   IF #_w5 AND ("DB_Data".F20.Sensor_Correct_Position OR ("DB_Data".F19.Sensor_Correct_Position AND NOT "DB_Data".F20.Btt_Down_Selected) OR ("DB_Data".F18.Sensor_Correct_Position AND NOT "DB_Data".F20.Btt_Down_Selected AND NOT "DB_Data".F19.Btt_Up_Selected AND NOT "DB_Data".F19.Btt_Down_Selected) OR ("DB_Data".F17.Sensor_Correct_Position AND NOT "DB_Data".F20.Btt_Down_Selected AND NOT "DB_Data".F19.Btt_Up_Selected AND NOT "DB_Data".F19.Btt_Down_Selected AND NOT "DB_Data".F18.Btt_Up_Selected AND NOT "DB_Data".F18.Btt_Down_Selected) OR ("DB_Data".F16.Sensor_Correct_Position AND NOT "DB_Data".F20.Btt_Down_Selected AND NOT "DB_Data".F19.Btt_Up_Selected AND NOT "DB_Data".F19.Btt_Down_Selected AND NOT "DB_Data".F18.Btt_Up_Selected AND NOT "DB_Data".F18.Btt_Down_Selected AND NOT "DB_Data".F17.Btt_Up_Selected AND NOT "DB_Data".F17.Btt_Down_Selected) OR ("DB_Data".F15.Sensor_Correct_Position AND NOT "DB_Data".F20.Btt_Down_Selected AND NOT "DB_Data".F19.Btt_Up_Selected AND NOT "DB_Data".F19.Btt_Down_Selected AND NOT "DB_Data".F18.Btt_Up_Selected AND NOT "DB_Data".F18.Btt_Down_Selected AND NOT "DB_Data".F17.Btt_Up_Selected AND NOT "DB_Data".F17.Btt_Down_Selected AND NOT "DB_Data".F16.Btt_Up_Selected AND NOT "DB_Data".F16.Btt_Down_Selected) OR ("DB_Data".F14.Sensor_Correct_Position AND NOT "DB_Data".F20.Btt_Down_Selected AND NOT "DB_Data".F19.Btt_Up_Selected AND NOT "DB_Data".F19.Btt_Down_Selected AND NOT "DB_Data".F18.Btt_Up_Selected AND NOT "DB_Data".F18.Btt_Down_Selected AND NOT "DB_Data".F17.Btt_Up_Selected AND NOT "DB_Data".F17.Btt_Down_Selected AND NOT "DB_Data".F16.Btt_Up_Selected AND NOT "DB_Data".F16.Btt_Down_Selected AND NOT "DB_Data".F15.Btt_Up_Selected AND NOT "DB_Data".F15.Btt_Down_Selected) OR ("DB_Data".F13.Sensor_Correct_Position AND NOT "DB_Data".F20.Btt_Down_Selected AND NOT "DB_Data".F19.Btt_Up_Selected AND NOT "DB_Data".F19.Btt_Down_Selected AND NOT "DB_Data".F18.Btt_Up_Selected AND NOT "DB_Data".F18.Btt_Down_Selected AND NOT "DB_Data".F17.Btt_Up_Selected AND NOT "DB_Data".F17.Btt_Down_Selected AND NOT "DB_Data".F16.Btt_Up_Selected AND NOT "DB_Data".F16.Btt_Down_Selected AND NOT "DB_Data".F15.Btt_Up_Selected AND NOT "DB_Data".F15.Btt_Down_Selected AND NOT "DB_Data".F14.Btt_Up_Selected AND NOT "DB_Data".F14.Btt_Down_Selected) OR ("DB_Data".F12.Sensor_Correct_Position AND NOT "DB_Data".F20.Btt_Down_Selected AND NOT "DB_Data".F19.Btt_Up_Selected AND NOT "DB_Data".F19.Btt_Down_Selected AND NOT "DB_Data".F18.Btt_Up_Selected AND NOT "DB_Data".F18.Btt_Down_Selected AND NOT "DB_Data".F17.Btt_Up_Selected AND NOT "DB_Data".F17.Btt_Down_Selected AND NOT "DB_Data".F16.Btt_Up_Selected AND NOT "DB_Data".F16.Btt_Down_Selected AND NOT "DB_Data".F15.Btt_Up_Selected AND NOT "DB_Data".F15.Btt_Down_Selected AND NOT "DB_Data".F14.Btt_Up_Selected AND NOT "DB_Data".F14.Btt_Down_Selected AND NOT "DB_Data".F13.Btt_Up_Selected AND NOT "DB_Data".F13.Btt_Down_Selected) OR ("DB_Data".F11.Sensor_Correct_Position AND NOT "DB_Data".F20.Btt_Down_Selected AND NOT "DB_Data".F19.Btt_Up_Selected AND NOT "DB_Data".F19.Btt_Down_Selected AND NOT "DB_Data".F18.Btt_Up_Selected AND NOT "DB_Data".F18.Btt_Down_Selected AND NOT "DB_Data".F17.Btt_Up_Selected AND NOT "DB_Data".F17.Btt_Down_Selected AND NOT "DB_Data".F16.Btt_Up_Selected AND NOT "DB_Data".F16.Btt_Down_Selected AND NOT "DB_Data".F15.Btt_Up_Selected AND NOT "DB_Data".F15.Btt_Down_Selected AND NOT "DB_Data".F14.Btt_Up_Selected AND NOT "DB_Data".F14.Btt_Down_Selected AND NOT "DB_Data".F13.Btt_Up_Selected AND NOT "DB_Data".F13.Btt_Down_Selected AND NOT "DB_Data".F12.Btt_Up_Selected AND NOT "DB_Data".F12.Btt_Down_Selected) OR ("DB_Data".F10.Sensor_Correct_Position AND NOT "DB_Data".F20.Btt_Down_Selected AND NOT "DB_Data".F19.Btt_Up_Selected AND NOT "DB_Data".F19.Btt_Down_Selected AND NOT "DB_Data".F18.Btt_Up_Selected AND NOT "DB_Data".F18.Btt_Down_Selected AND NOT "DB_Data".F17.Btt_Up_Selected AND NOT "DB_Data".F17.Btt_Down_Selected AND NOT "DB_Data".F16.Btt_Up_Selected AND NOT "DB_Data".F16.Btt_Down_Selected AND NOT "DB_Data".F15.Btt_Up_Selected AND NOT "DB_Data".F15.Btt_Down_Selected AND NOT "DB_Data".F14.Btt_Up_Selected AND NOT "DB_Data".F14.Btt_Down_Selected AND NOT "DB_Data".F13.Btt_Up_Selected AND NOT "DB_Data".F13.Btt_Down_Selected AND NOT "DB_Data".F12.Btt_Up_Selected AND NOT "DB_Data".F12.Btt_Down_Selected AND NOT "DB_Data".F11.Btt_Up_Selected AND NOT "DB_Data".F11.Btt_Down_Selected) OR ("DB_Data".F9.Sensor_Correct_Position AND NOT "DB_Data".F20.Btt_Down_Selected AND NOT "DB_Data".F19.Btt_Up_Selected AND NOT "DB_Data".F19.Btt_Down_Selected AND NOT "DB_Data".F18.Btt_Up_Selected AND NOT "DB_Data".F18.Btt_Down_Selected AND NOT "DB_Data".F17.Btt_Up_Selected AND NOT "DB_Data".F17.Btt_Down_Selected AND NOT "DB_Data".F16.Btt_Up_Selected AND NOT "DB_Data".F16.Btt_Down_Selected AND NOT "DB_Data".F15.Btt_Up_Selected AND NOT "DB_Data".F15.Btt_Down_Selected AND NOT "DB_Data".F14.Btt_Up_Selected AND NOT "DB_Data".F14.Btt_Down_Selected AND NOT "DB_Data".F13.Btt_Up_Selected AND NOT "DB_Data".F13.Btt_Down_Selected AND NOT "DB_Data".F12.Btt_Up_Selected AND NOT "DB_Data".F12.Btt_Down_Selected AND NOT "DB_Data".F11.Btt_Up_Selected AND NOT "DB_Data".F11.Btt_Down_Selected AND NOT "DB_Data".F10.Btt_Up_Selected AND NOT "DB_Data".F10.Btt_Down_Selected) OR ("DB_Data".F8.Sensor_Correct_Position AND NOT "DB_Data".F20.Btt_Down_Selected AND NOT "DB_Data".F19.Btt_Up_Selected AND NOT "DB_Data".F19.Btt_Down_Selected AND NOT "DB_Data".F18.Btt_Up_Selected AND NOT "DB_Data".F18.Btt_Down_Selected AND NOT "DB_Data".F17.Btt_Up_Selected AND NOT "DB_Data".F17.Btt_Down_Selected AND NOT "DB_Data".F16.Btt_Up_Selected AND NOT "DB_Data".F16.Btt_Down_Selected AND NOT "DB_Data".F15.Btt_Up_Selected AND NOT "DB_Data".F15.Btt_Down_Selected AND NOT "DB_Data".F14.Btt_Up_Selected AND NOT "DB_Data".F14.Btt_Down_Selected AND NOT "DB_Data".F13.Btt_Up_Selected AND NOT "DB_Data".F13.Btt_Down_Selected AND NOT "DB_Data".F12.Btt_Up_Selected AND NOT "DB_Data".F12.Btt_Down_Selected AND NOT "DB_Data".F11.Btt_Up_Selected AND NOT "DB_Data".F11.Btt_Down_Selected AND NOT "DB_Data".F10.Btt_Up_Selected AND NOT "DB_Data".F10.Btt_Down_Selected AND NOT "DB_Data".F9.Btt_Up_Selected AND NOT "DB_Data".F9.Btt_Down_Selected) OR ("DB_Data".F7.Sensor_Correct_Position AND NOT "DB_Data".F20.Btt_Down_Selected AND NOT "DB_Data".F19.Btt_Up_Selected AND NOT "DB_Data".F19.Btt_Down_Selected AND NOT "DB_Data".F18.Btt_Up_Selected AND NOT "DB_Data".F18.Btt_Down_Selected AND NOT "DB_Data".F17.Btt_Up_Selected AND NOT "DB_Data".F17.Btt_Down_Selected AND NOT "DB_Data".F16.Btt_Up_Selected AND NOT "DB_Data".F16.Btt_Down_Selected AND NOT "DB_Data".F15.Btt_Up_Selected AND NOT "DB_Data".F15.Btt_Down_Selected AND NOT "DB_Data".F14.Btt_Up_Selected AND NOT "DB_Data".F14.Btt_Down_Selected AND NOT "DB_Data".F13.Btt_Up_Selected AND NOT "DB_Data".F13.Btt_Down_Selected AND NOT "DB_Data".F12.Btt_Up_Selected AND NOT "DB_Data".F12.Btt_Down_Selected AND NOT "DB_Data".F11.Btt_Up_Selected AND NOT "DB_Data".F11.Btt_Down_Selected AND NOT "DB_Data".F10.Btt_Up_Selected AND NOT "DB_Data".F10.Btt_Down_Selected AND NOT "DB_Data".F9.Btt_Up_Selected AND NOT "DB_Data".F9.Btt_Down_Selected AND NOT "DB_Data".F8.Btt_Up_Selected AND NOT "DB_Data".F8.Btt_Down_Selected) OR ("DB_Data".F6.Sensor_Correct_Position AND NOT "DB_Data".F20.Btt_Down_Selected AND NOT "DB_Data".F19.Btt_Up_Selected AND NOT "DB_Data".F19.Btt_Down_Selected AND NOT "DB_Data".F18.Btt_Up_Selected AND NOT "DB_Data".F18.Btt_Down_Selected AND NOT "DB_Data".F17.Btt_Up_Selected AND NOT "DB_Data".F17.Btt_Down_Selected AND NOT "DB_Data".F16.Btt_Up_Selected AND NOT "DB_Data".F16.Btt_Down_Selected AND NOT "DB_Data".F15.Btt_Up_Selected AND NOT "DB_Data".F15.Btt_Down_Selected AND NOT "DB_Data".F14.Btt_Up_Selected AND NOT "DB_Data".F14.Btt_Down_Selected AND NOT "DB_Data".F13.Btt_Up_Selected AND NOT "DB_Data".F13.Btt_Down_Selected AND NOT "DB_Data".F12.Btt_Up_Selected AND NOT "DB_Data".F12.Btt_Down_Selected AND NOT "DB_Data".F11.Btt_Up_Selected AND NOT "DB_Data".F11.Btt_Down_Selected AND NOT "DB_Data".F10.Btt_Up_Selected AND NOT "DB_Data".F10.Btt_Down_Selected AND NOT "DB_Data".F9.Btt_Up_Selected AND NOT "DB_Data".F9.Btt_Down_Selected AND NOT "DB_Data".F8.Btt_Up_Selected AND NOT "DB_Data".F8.Btt_Down_Selected AND NOT "DB_Data".F7.Btt_Up_Selected AND NOT "DB_Data".F7.Btt_Down_Selected) OR ("DB_Data".F5.Sensor_Correct_Position AND NOT "DB_Data".F20.Btt_Down_Selected AND NOT "DB_Data".F19.Btt_Up_Selected AND NOT "DB_Data".F19.Btt_Down_Selected AND NOT "DB_Data".F18.Btt_Up_Selected AND NOT "DB_Data".F18.Btt_Down_Selected AND NOT "DB_Data".F17.Btt_Up_Selected AND NOT "DB_Data".F17.Btt_Down_Selected AND NOT "DB_Data".F16.Btt_Up_Selected AND NOT "DB_Data".F16.Btt_Down_Selected AND NOT "DB_Data".F15.Btt_Up_Selected AND NOT "DB_Data".F15.Btt_Down_Selected AND NOT "DB_Data".F14.Btt_Up_Selected AND NOT "DB_Data".F14.Btt_Down_Selected AND NOT "DB_Data".F13.Btt_Up_Selected AND NOT "DB_Data".F13.Btt_Down_Selected AND NOT "DB_Data".F12.Btt_Up_Selected AND NOT "DB_Data".F12.Btt_Down_Selected AND NOT "DB_Data".F11.Btt_Up_Selected AND NOT "DB_Data".F11.Btt_Down_Selected AND NOT "DB_Data".F10.Btt_Up_Selected AND NOT "DB_Data".F10.Btt_Down_Selected AND NOT "DB_Data".F9.Btt_Up_Selected AND NOT "DB_Data".F9.Btt_Down_Selected AND NOT "DB_Data".F8.Btt_Up_Selected AND NOT "DB_Data".F8.Btt_Down_Selected AND NOT "DB_Data".F7.Btt_Up_Selected AND NOT "DB_Data".F7.Btt_Down_Selected AND NOT "DB_Data".F6.Btt_Up_Selected AND NOT "DB_Data".F6.Btt_Down_Selected) OR ("DB_Data".F4.Sensor_Correct_Position AND NOT "DB_Data".F20.Btt_Down_Selected AND NOT "DB_Data".F19.Btt_Up_Selected AND NOT "DB_Data".F19.Btt_Down_Selected AND NOT "DB_Data".F18.Btt_Up_Selected AND NOT "DB_Data".F18.Btt_Down_Selected AND NOT "DB_Data".F17.Btt_Up_Selected AND NOT "DB_Data".F17.Btt_Down_Selected AND NOT "DB_Data".F16.Btt_Up_Selected AND NOT "DB_Data".F16.Btt_Down_Selected AND NOT "DB_Data".F15.Btt_Up_Selected AND NOT "DB_Data".F15.Btt_Down_Selected AND NOT "DB_Data".F14.Btt_Up_Selected AND NOT "DB_Data".F14.Btt_Down_Selected AND NOT "DB_Data".F13.Btt_Up_Selected AND NOT "DB_Data".F13.Btt_Down_Selected AND NOT "DB_Data".F12.Btt_Up_Selected AND NOT "DB_Data".F12.Btt_Down_Selected AND NOT "DB_Data".F11.Btt_Up_Selected AND NOT "DB_Data".F11.Btt_Down_Selected AND NOT "DB_Data".F10.Btt_Up_Selected AND NOT "DB_Data".F10.Btt_Down_Selected AND NOT "DB_Data".F9.Btt_Up_Selected AND NOT "DB_Data".F9.Btt_Down_Selected AND NOT "DB_Data".F8.Btt_Up_Selected AND NOT "DB_Data".F8.Btt_Down_Selected AND NOT "DB_Data".F7.Btt_Up_Selected AND NOT "DB_Data".F7.Btt_Down_Selected AND NOT "DB_Data".F6.Btt_Up_Selected AND NOT "DB_Data".F6.Btt_Down_Selected AND NOT "DB_Data".F5.Btt_Up_Selected AND NOT "DB_Data".F5.Btt_Down_Selected) OR ("DB_Data".F3.Sensor_Correct_Position AND NOT "DB_Data".F20.Btt_Down_Selected AND NOT "DB_Data".F19.Btt_Up_Selected AND NOT "DB_Data".F19.Btt_Down_Selected AND NOT "DB_Data".F18.Btt_Up_Selected AND NOT "DB_Data".F18.Btt_Down_Selected AND NOT "DB_Data".F17.Btt_Up_Selected AND NOT "DB_Data".F17.Btt_Down_Selected AND NOT "DB_Data".F16.Btt_Up_Selected AND NOT "DB_Data".F16.Btt_Down_Selected AND NOT "DB_Data".F15.Btt_Up_Selected AND NOT "DB_Data".F15.Btt_Down_Selected AND NOT "DB_Data".F14.Btt_Up_Selected AND NOT "DB_Data".F14.Btt_Down_Selected AND NOT "DB_Data".F13.Btt_Up_Selected AND NOT "DB_Data".F13.Btt_Down_Selected AND NOT "DB_Data".F12.Btt_Up_Selected AND NOT "DB_Data".F12.Btt_Down_Selected AND NOT "DB_Data".F11.Btt_Up_Selected AND NOT "DB_Data".F11.Btt_Down_Selected AND NOT "DB_Data".F10.Btt_Up_Selected AND NOT "DB_Data".F10.Btt_Down_Selected AND NOT "DB_Data".F9.Btt_Up_Selected AND NOT "DB_Data".F9.Btt_Down_Selected AND NOT "DB_Data".F8.Btt_Up_Selected AND NOT "DB_Data".F8.Btt_Down_Selected AND NOT "DB_Data".F7.Btt_Up_Selected AND NOT "DB_Data".F7.Btt_Down_Selected AND NOT "DB_Data".F6.Btt_Up_Selected AND NOT "DB_Data".F6.Btt_Down_Selected AND NOT "DB_Data".F5.Btt_Up_Selected AND NOT "DB_Data".F5.Btt_Down_Selected AND NOT "DB_Data".F4.Btt_Up_Selected AND NOT "DB_Data".F4.Btt_Down_Selected) OR ("DB_Data".F2.Sensor_Correct_Position AND NOT "DB_Data".F20.Btt_Down_Selected AND NOT "DB_Data".F19.Btt_Up_Selected AND NOT "DB_Data".F19.Btt_Down_Selected AND NOT "DB_Data".F18.Btt_Up_Selected AND NOT "DB_Data".F18.Btt_Down_Selected AND NOT "DB_Data".F17.Btt_Up_Selected AND NOT "DB_Data".F17.Btt_Down_Selected AND NOT "DB_Data".F16.Btt_Up_Selected AND NOT "DB_Data".F16.Btt_Down_Selected AND NOT "DB_Data".F15.Btt_Up_Selected AND NOT "DB_Data".F15.Btt_Down_Selected AND NOT "DB_Data".F14.Btt_Up_Selected AND NOT "DB_Data".F14.Btt_Down_Selected AND NOT "DB_Data".F13.Btt_Up_Selected AND NOT "DB_Data".F13.Btt_Down_Selected AND NOT "DB_Data".F12.Btt_Up_Selected AND NOT "DB_Data".F12.Btt_Down_Selected AND NOT "DB_Data".F11.Btt_Up_Selected AND NOT "DB_Data".F11.Btt_Down_Selected AND NOT "DB_Data".F10.Btt_Up_Selected AND NOT "DB_Data".F10.Btt_Down_Selected AND NOT "DB_Data".F9.Btt_Up_Selected AND NOT "DB_Data".F9.Btt_Down_Selected AND NOT "DB_Data".F8.Btt_Up_Selected AND NOT "DB_Data".F8.Btt_Down_Selected AND NOT "DB_Data".F7.Btt_Up_Selected AND NOT "DB_Data".F7.Btt_Down_Selected AND NOT "DB_Data".F6.Btt_Up_Selected AND NOT "DB_Data".F6.Btt_Down_Selected AND NOT "DB_Data".F5.Btt_Up_Selected AND NOT "DB_Data".F5.Btt_Down_Selected AND NOT "DB_Data".F4.Btt_Up_Selected AND NOT "DB_Data".F4.Btt_Down_Selected AND NOT "DB_Data".F3.Btt_Down_Selected AND NOT "DB_Data".F3.Btt_Up_Selected) OR ("DB_Data".F1.Sensor_Correct_Position AND NOT "DB_Data".F20.Btt_Down_Selected AND NOT "DB_Data".F19.Btt_Up_Selected AND NOT "DB_Data".F19.Btt_Down_Selected AND NOT "DB_Data".F18.Btt_Up_Selected AND NOT "DB_Data".F18.Btt_Down_Selected AND NOT "DB_Data".F17.Btt_Up_Selected AND NOT "DB_Data".F17.Btt_Down_Selected AND NOT "DB_Data".F16.Btt_Up_Selected AND NOT "DB_Data".F16.Btt_Down_Selected AND NOT "DB_Data".F15.Btt_Up_Selected AND NOT "DB_Data".F15.Btt_Down_Selected AND NOT "DB_Data".F14.Btt_Up_Selected AND NOT "DB_Data".F14.Btt_Down_Selected AND NOT "DB_Data".F13.Btt_Up_Selected AND NOT "DB_Data".F13.Btt_Down_Selected AND NOT "DB_Data".F12.Btt_Up_Selected AND NOT "DB_Data".F12.Btt_Down_Selected AND NOT "DB_Data".F11.Btt_Up_Selected AND NOT "DB_Data".F11.Btt_Down_Selected AND NOT "DB_Data".F10.Btt_Up_Selected AND NOT "DB_Data".F10.Btt_Down_Selected AND NOT "DB_Data".F9.Btt_Up_Selected AND NOT "DB_Data".F9.Btt_Down_Selected AND NOT "DB_Data".F8.Btt_Up_Selected AND NOT "DB_Data".F8.Btt_Down_Selected AND NOT "DB_Data".F7.Btt_Up_Selected AND NOT "DB_Data".F7.Btt_Down_Selected AND NOT "DB_Data".F6.Btt_Up_Selected AND NOT "DB_Data".F6.Btt_Down_Selected AND NOT "DB_Data".F5.Btt_Up_Selected AND NOT "DB_Data".F5.Btt_Down_Selected AND NOT "DB_Data".F4.Btt_Up_Selected AND NOT "DB_Data".F4.Btt_Down_Selected AND NOT "DB_Data".F3.Btt_Down_Selected AND NOT "DB_Data".F3.Btt_Up_Selected AND NOT "DB_Data".F2.Btt_Down_Selected AND NOT "DB_Data".F2.Btt_Up_Selected)) THEN
       "DB_Data".Last_Is_Up := FALSE;
   END_IF;
END_REGION

REGION Network 23
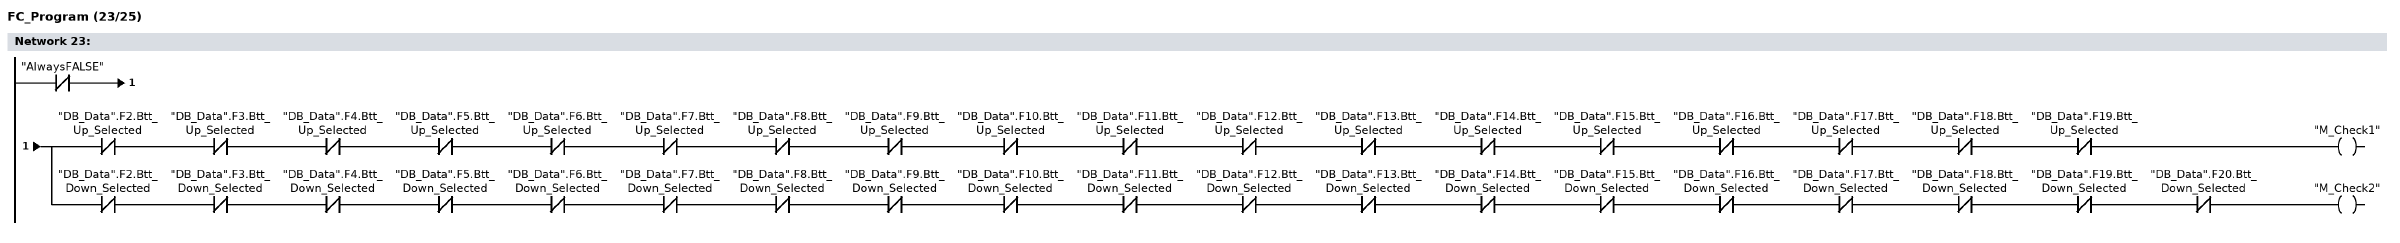
   RUNG wire#powerrail
      I_Contact( "AlwaysFALSE" )
      wire#w1
      I_Contact( "DB_Data".F2.Btt_Up_Selected )
      I_Contact( "DB_Data".F3.Btt_Up_Selected )
      I_Contact( "DB_Data".F4.Btt_Up_Selected )
      I_Contact( "DB_Data".F5.Btt_Up_Selected )
      I_Contact( "DB_Data".F6.Btt_Up_Selected )
      I_Contact( "DB_Data".F7.Btt_Up_Selected )
      I_Contact( "DB_Data".F8.Btt_Up_Selected )
      I_Contact( "DB_Data".F9.Btt_Up_Selected )
      I_Contact( "DB_Data".F10.Btt_Up_Selected )
      I_Contact( "DB_Data".F11.Btt_Up_Selected )
      I_Contact( "DB_Data".F12.Btt_Up_Selected )
      I_Contact( "DB_Data".F13.Btt_Up_Selected )
      I_Contact( "DB_Data".F14.Btt_Up_Selected )
      I_Contact( "DB_Data".F15.Btt_Up_Selected )
      I_Contact( "DB_Data".F16.Btt_Up_Selected )
      I_Contact( "DB_Data".F17.Btt_Up_Selected )
      I_Contact( "DB_Data".F18.Btt_Up_Selected )
      I_Contact( "DB_Data".F19.Btt_Up_Selected )
      Coil( "M_Check1" )
   END_RUNG
   RUNG wire#w1
      I_Contact( "DB_Data".F2.Btt_Down_Selected )
      I_Contact( "DB_Data".F3.Btt_Down_Selected )
      I_Contact( "DB_Data".F4.Btt_Down_Selected )
      I_Contact( "DB_Data".F5.Btt_Down_Selected )
      I_Contact( "DB_Data".F6.Btt_Down_Selected )
      I_Contact( "DB_Data".F7.Btt_Down_Selected )
      I_Contact( "DB_Data".F8.Btt_Down_Selected )
      I_Contact( "DB_Data".F9.Btt_Down_Selected )
      I_Contact( "DB_Data".F10.Btt_Down_Selected )
      I_Contact( "DB_Data".F11.Btt_Down_Selected )
      I_Contact( "DB_Data".F12.Btt_Down_Selected )
      I_Contact( "DB_Data".F13.Btt_Down_Selected )
      I_Contact( "DB_Data".F14.Btt_Down_Selected )
      I_Contact( "DB_Data".F15.Btt_Down_Selected )
      I_Contact( "DB_Data".F16.Btt_Down_Selected )
      I_Contact( "DB_Data".F17.Btt_Down_Selected )
      I_Contact( "DB_Data".F18.Btt_Down_Selected )
      I_Contact( "DB_Data".F19.Btt_Down_Selected )
      I_Contact( "DB_Data".F20.Btt_Down_Selected )
      Coil( "M_Check2" )
   END_RUNG
   // the same network as SCL:
   "M_Check1" := NOT "AlwaysFALSE" AND NOT "DB_Data".F2.Btt_Up_Selected AND NOT "DB_Data".F3.Btt_Up_Selected AND NOT "DB_Data".F4.Btt_Up_Selected AND NOT "DB_Data".F5.Btt_Up_Selected AND NOT "DB_Data".F6.Btt_Up_Selected AND NOT "DB_Data".F7.Btt_Up_Selected AND NOT "DB_Data".F8.Btt_Up_Selected AND NOT "DB_Data".F9.Btt_Up_Selected AND NOT "DB_Data".F10.Btt_Up_Selected AND NOT "DB_Data".F11.Btt_Up_Selected AND NOT "DB_Data".F12.Btt_Up_Selected AND NOT "DB_Data".F13.Btt_Up_Selected AND NOT "DB_Data".F14.Btt_Up_Selected AND NOT "DB_Data".F15.Btt_Up_Selected AND NOT "DB_Data".F16.Btt_Up_Selected AND NOT "DB_Data".F17.Btt_Up_Selected AND NOT "DB_Data".F18.Btt_Up_Selected AND NOT "DB_Data".F19.Btt_Up_Selected;
   "M_Check2" := NOT "AlwaysFALSE" AND NOT "DB_Data".F2.Btt_Down_Selected AND NOT "DB_Data".F3.Btt_Down_Selected AND NOT "DB_Data".F4.Btt_Down_Selected AND NOT "DB_Data".F5.Btt_Down_Selected AND NOT "DB_Data".F6.Btt_Down_Selected AND NOT "DB_Data".F7.Btt_Down_Selected AND NOT "DB_Data".F8.Btt_Down_Selected AND NOT "DB_Data".F9.Btt_Down_Selected AND NOT "DB_Data".F10.Btt_Down_Selected AND NOT "DB_Data".F11.Btt_Down_Selected AND NOT "DB_Data".F12.Btt_Down_Selected AND NOT "DB_Data".F13.Btt_Down_Selected AND NOT "DB_Data".F14.Btt_Down_Selected AND NOT "DB_Data".F15.Btt_Down_Selected AND NOT "DB_Data".F16.Btt_Down_Selected AND NOT "DB_Data".F17.Btt_Down_Selected AND NOT "DB_Data".F18.Btt_Down_Selected AND NOT "DB_Data".F19.Btt_Down_Selected AND NOT "DB_Data".F20.Btt_Down_Selected;
END_REGION

REGION Network 24: Tự động mở cửa
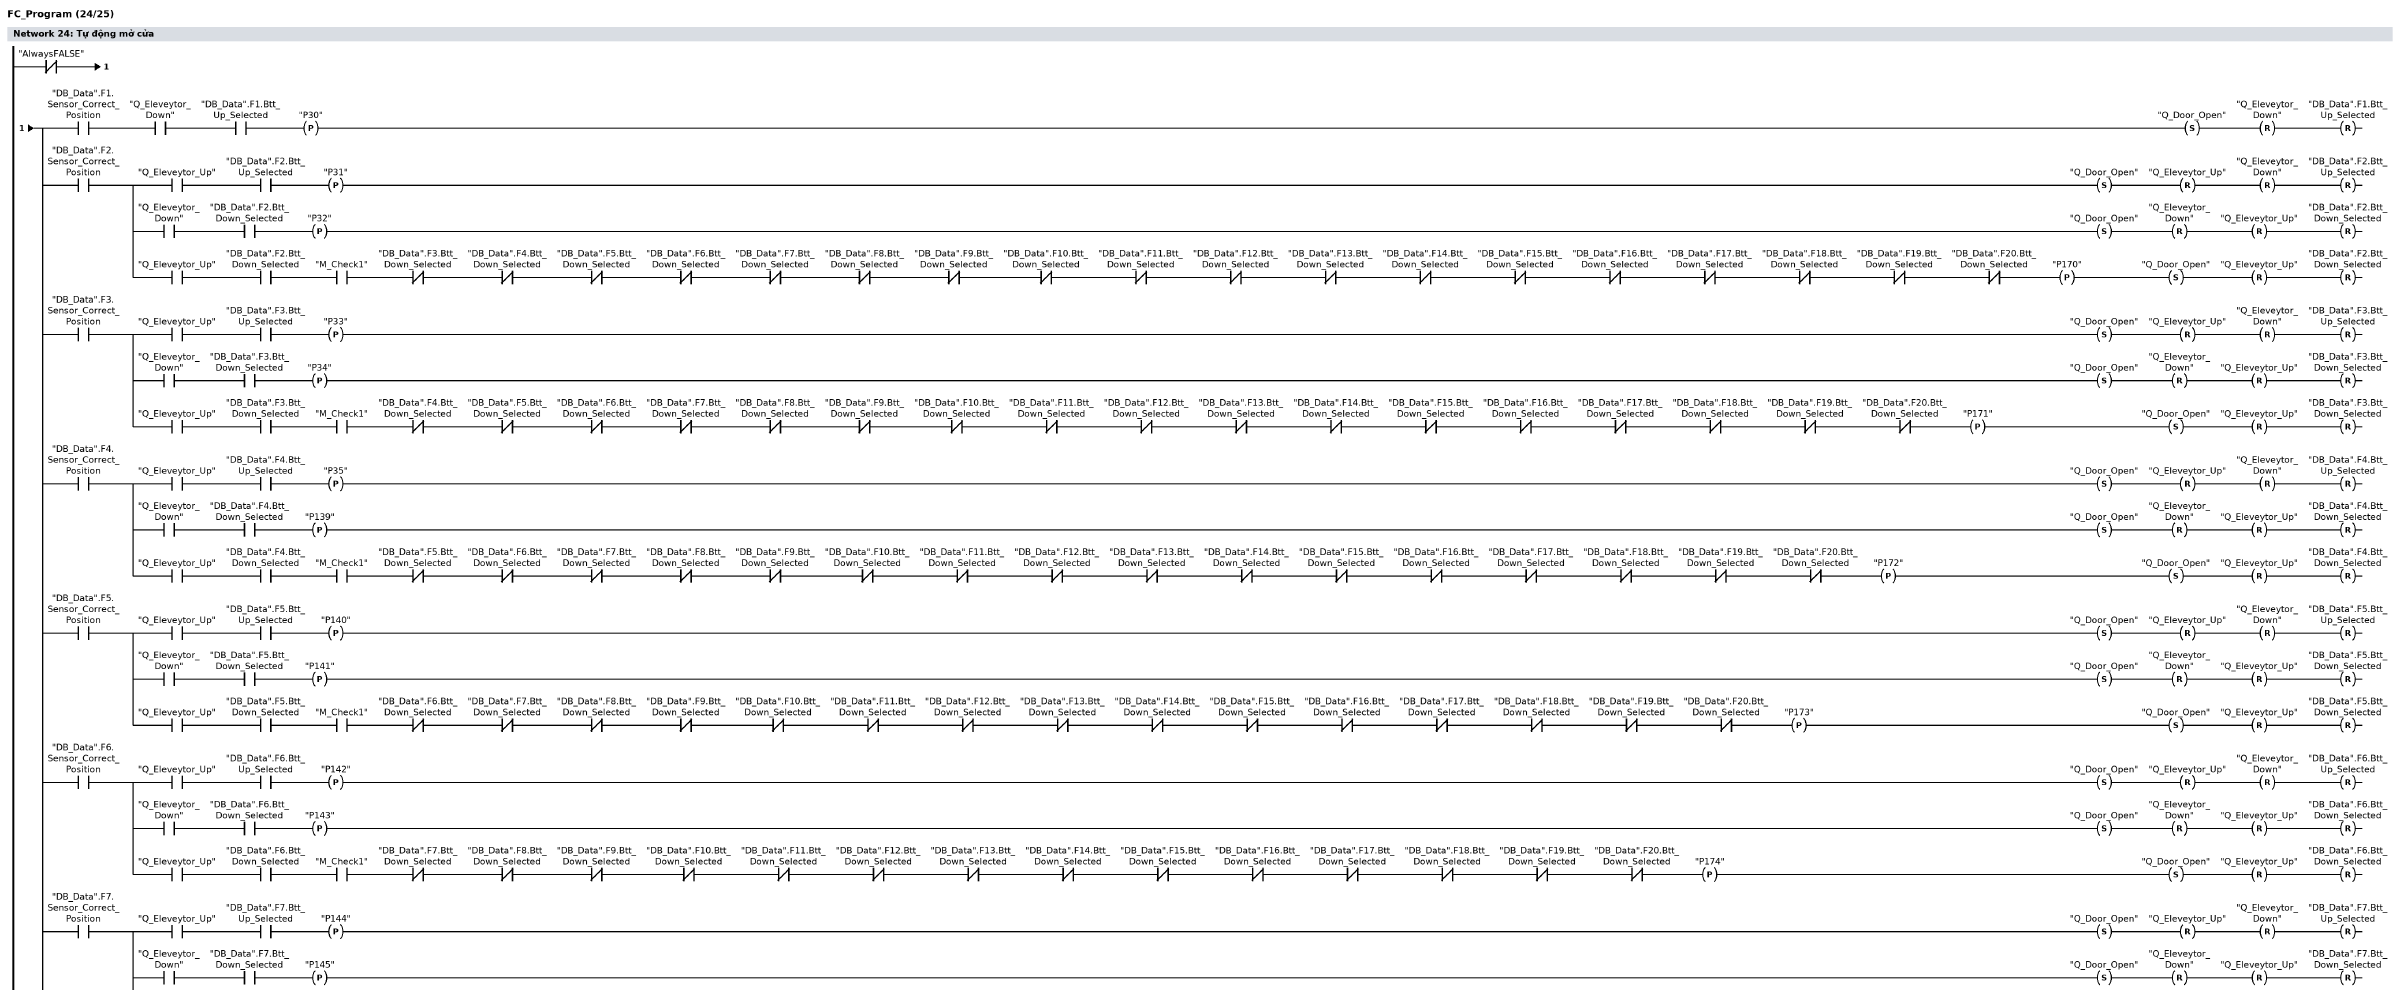
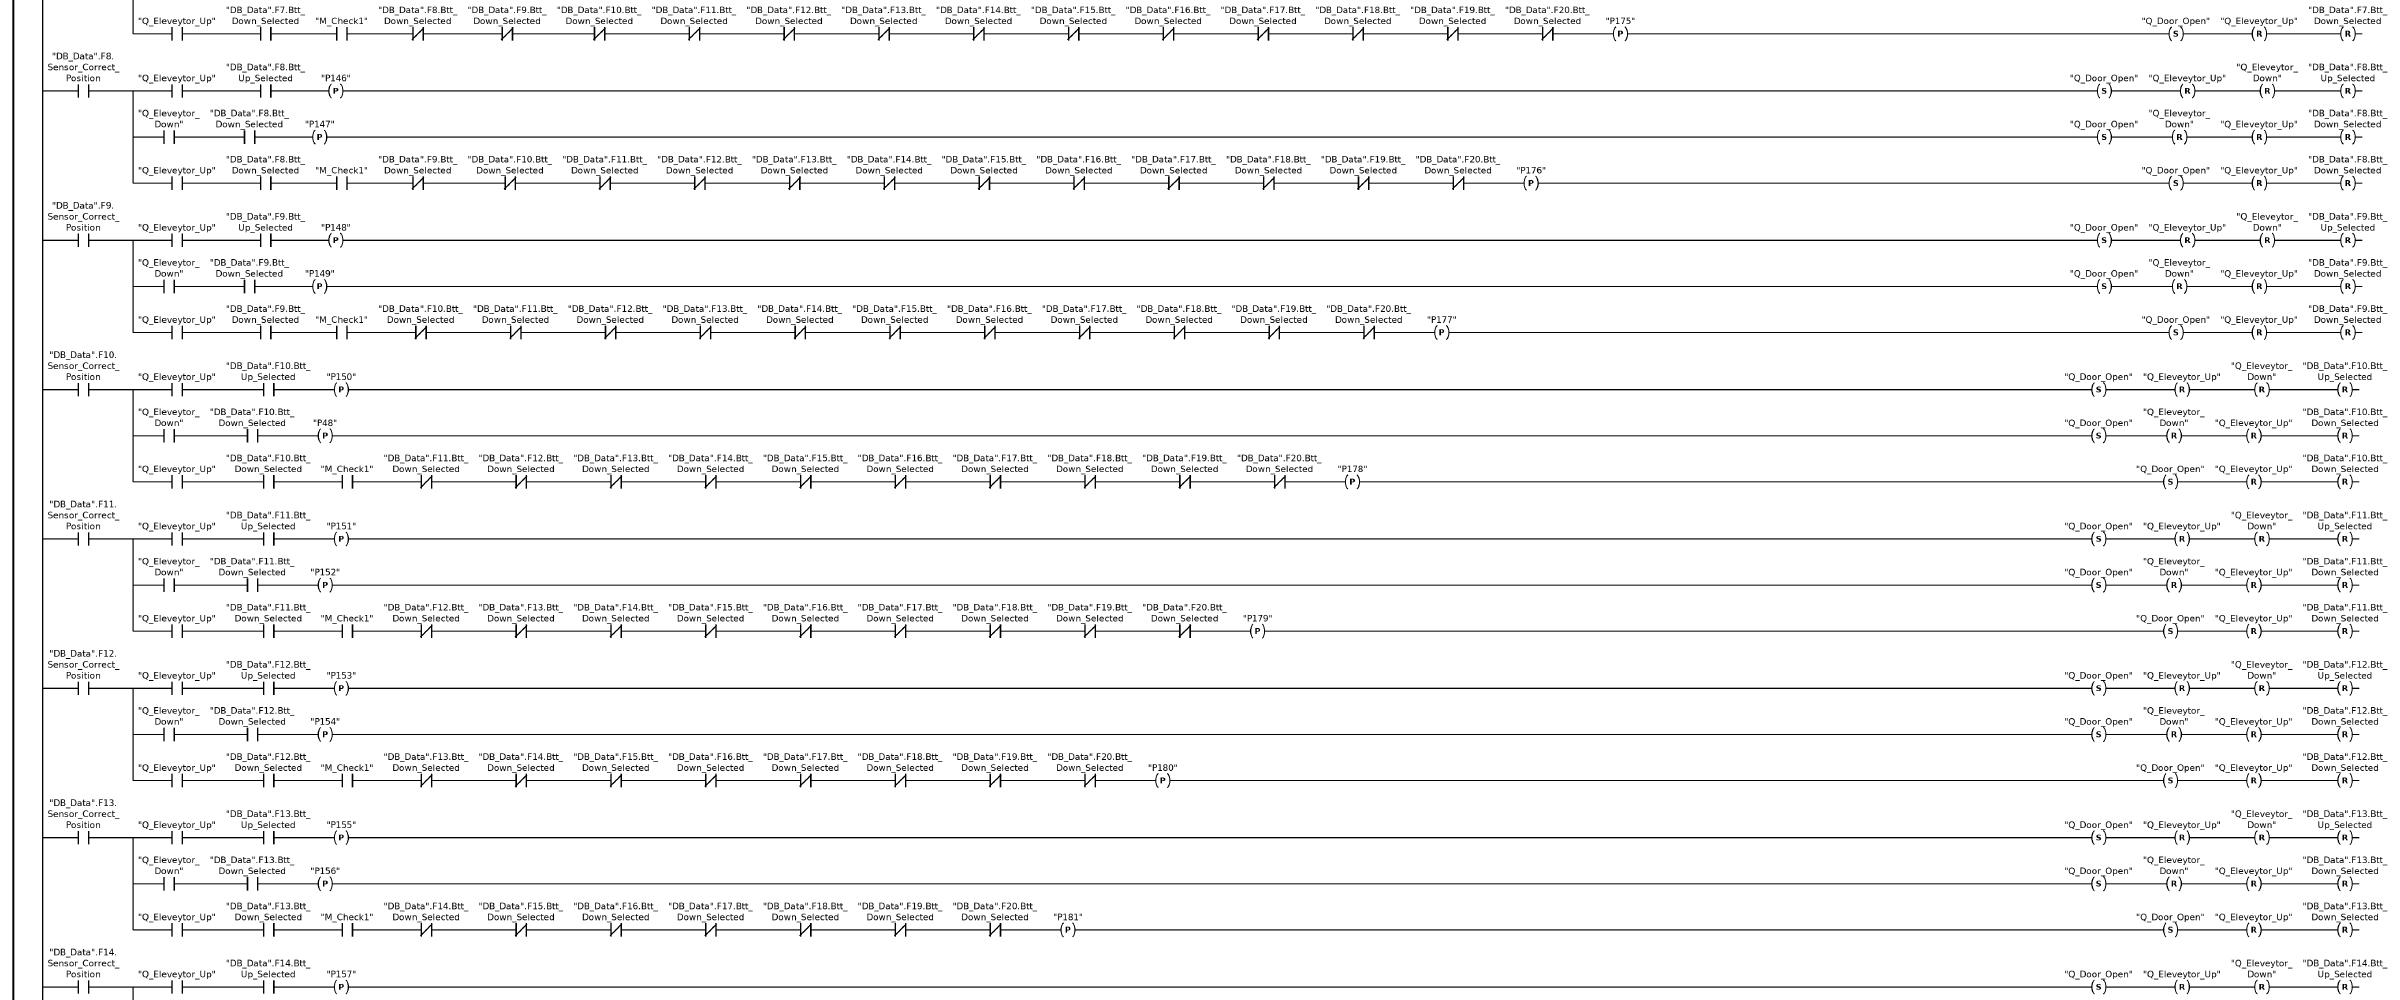
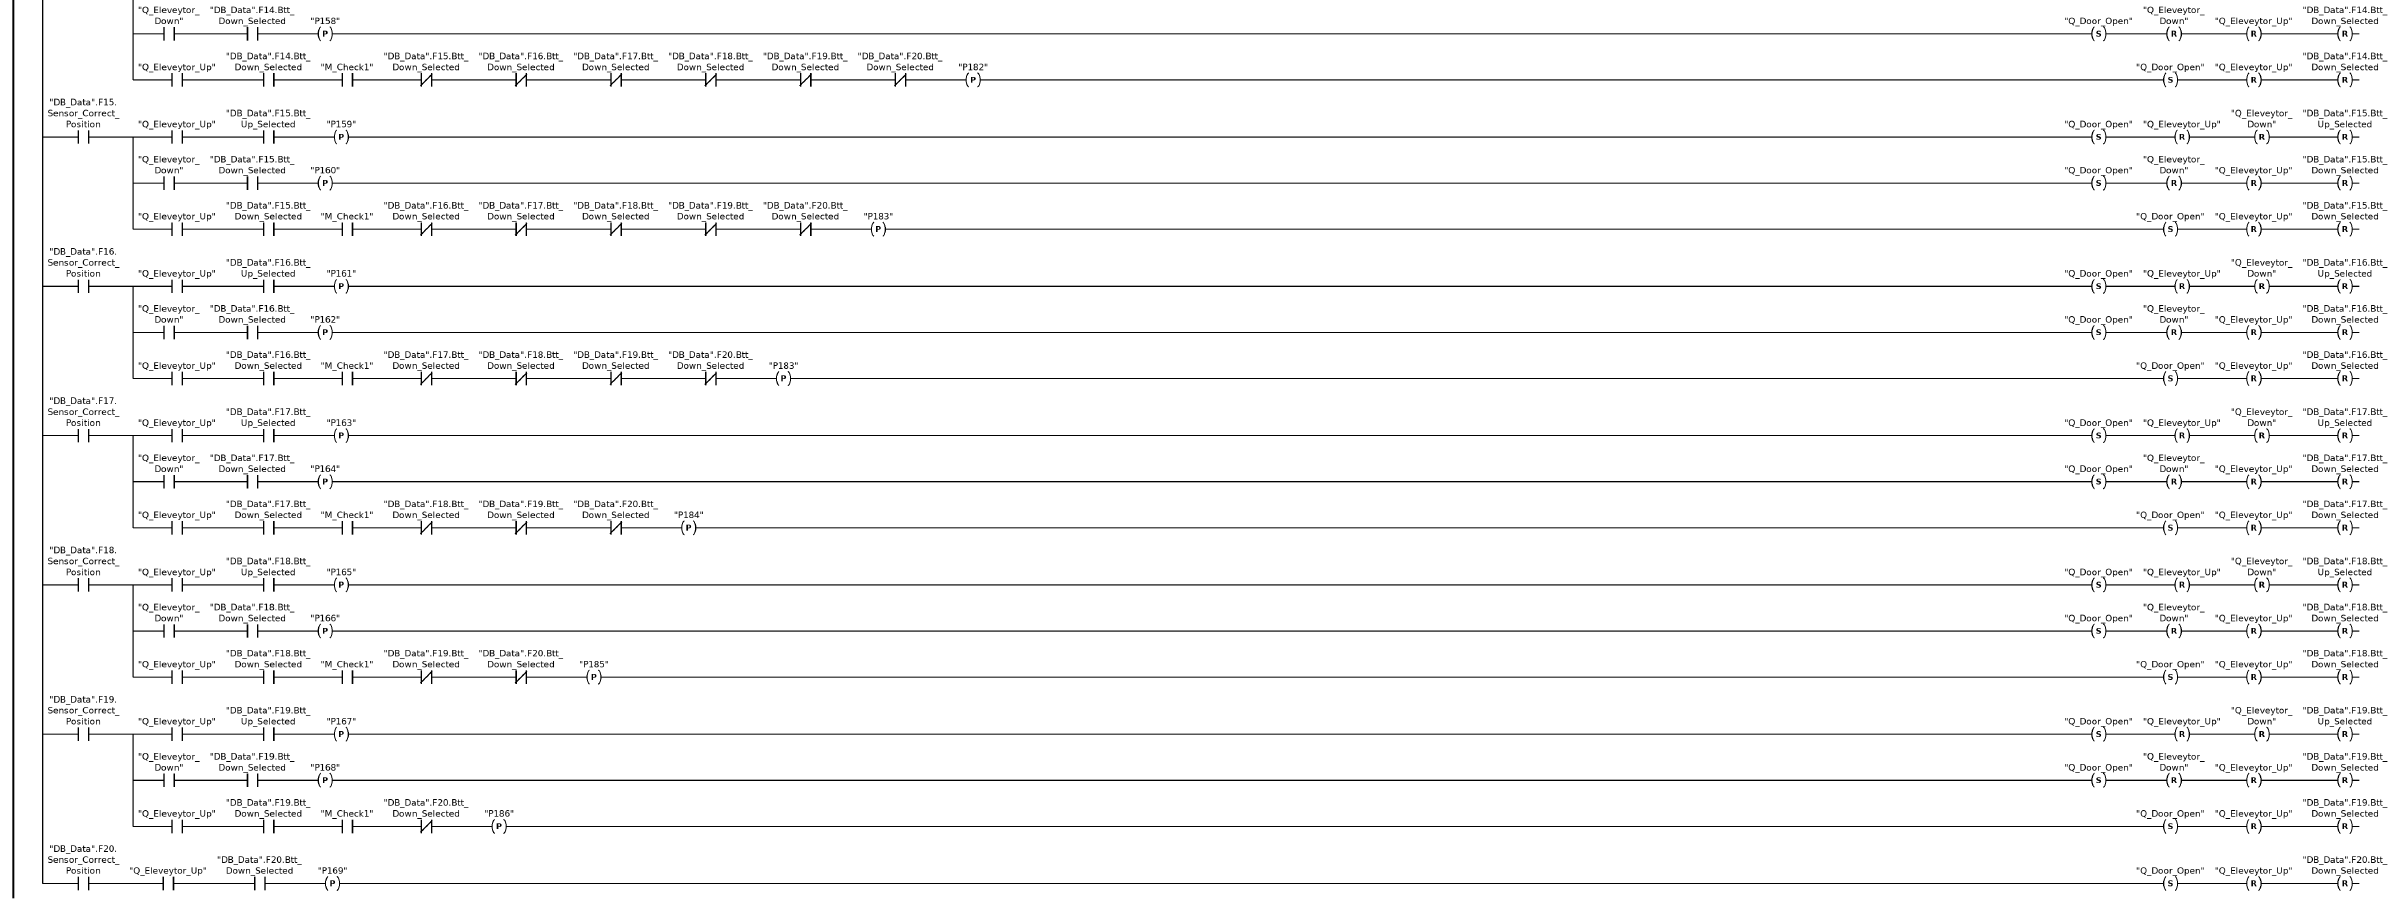
   RUNG wire#powerrail
      I_Contact( "AlwaysFALSE" )
      wire#w1
      Contact( "DB_Data".F1.Sensor_Correct_Position )
      Contact( "Q_Eleveytor_Down" )
      Contact( "DB_Data".F1.Btt_Up_Selected )
      P_Trig( "P30" )
      S_Coil( "Q_Door_Open" )
      R_Coil( "Q_Eleveytor_Down" )
      R_Coil( "DB_Data".F1.Btt_Up_Selected )
   END_RUNG
   RUNG wire#w1
      Contact( "DB_Data".F2.Sensor_Correct_Position )
      wire#w2
      Contact( "Q_Eleveytor_Up" )
      Contact( "DB_Data".F2.Btt_Up_Selected )
      P_Trig( "P31" )
      S_Coil( "Q_Door_Open" )
      R_Coil( "Q_Eleveytor_Up" )
      R_Coil( "Q_Eleveytor_Down" )
      R_Coil( "DB_Data".F2.Btt_Up_Selected )
   END_RUNG
   RUNG wire#w2
      Contact( "Q_Eleveytor_Down" )
      Contact( "DB_Data".F2.Btt_Down_Selected )
      P_Trig( "P32" )
      S_Coil( "Q_Door_Open" )
      R_Coil( "Q_Eleveytor_Down" )
      R_Coil( "Q_Eleveytor_Up" )
      R_Coil( "DB_Data".F2.Btt_Down_Selected )
   END_RUNG
   RUNG wire#w2
      Contact( "Q_Eleveytor_Up" )
      Contact( "DB_Data".F2.Btt_Down_Selected )
      Contact( "M_Check1" )
      I_Contact( "DB_Data".F3.Btt_Down_Selected )
      I_Contact( "DB_Data".F4.Btt_Down_Selected )
      I_Contact( "DB_Data".F5.Btt_Down_Selected )
      I_Contact( "DB_Data".F6.Btt_Down_Selected )
      I_Contact( "DB_Data".F7.Btt_Down_Selected )
      I_Contact( "DB_Data".F8.Btt_Down_Selected )
      I_Contact( "DB_Data".F9.Btt_Down_Selected )
      I_Contact( "DB_Data".F10.Btt_Down_Selected )
      I_Contact( "DB_Data".F11.Btt_Down_Selected )
      I_Contact( "DB_Data".F12.Btt_Down_Selected )
      I_Contact( "DB_Data".F13.Btt_Down_Selected )
      I_Contact( "DB_Data".F14.Btt_Down_Selected )
      I_Contact( "DB_Data".F15.Btt_Down_Selected )
      I_Contact( "DB_Data".F16.Btt_Down_Selected )
      I_Contact( "DB_Data".F17.Btt_Down_Selected )
      I_Contact( "DB_Data".F18.Btt_Down_Selected )
      I_Contact( "DB_Data".F19.Btt_Down_Selected )
      I_Contact( "DB_Data".F20.Btt_Down_Selected )
      P_Trig( "P170" )
      S_Coil( "Q_Door_Open" )
      R_Coil( "Q_Eleveytor_Up" )
      R_Coil( "DB_Data".F2.Btt_Down_Selected )
   END_RUNG
   RUNG wire#w1
      Contact( "DB_Data".F3.Sensor_Correct_Position )
      wire#w3
      Contact( "Q_Eleveytor_Up" )
      Contact( "DB_Data".F3.Btt_Up_Selected )
      P_Trig( "P33" )
      S_Coil( "Q_Door_Open" )
      R_Coil( "Q_Eleveytor_Up" )
      R_Coil( "Q_Eleveytor_Down" )
      R_Coil( "DB_Data".F3.Btt_Up_Selected )
   END_RUNG
   RUNG wire#w3
      Contact( "Q_Eleveytor_Down" )
      Contact( "DB_Data".F3.Btt_Down_Selected )
      P_Trig( "P34" )
      S_Coil( "Q_Door_Open" )
      R_Coil( "Q_Eleveytor_Down" )
      R_Coil( "Q_Eleveytor_Up" )
      R_Coil( "DB_Data".F3.Btt_Down_Selected )
   END_RUNG
   RUNG wire#w3
      Contact( "Q_Eleveytor_Up" )
      Contact( "DB_Data".F3.Btt_Down_Selected )
      Contact( "M_Check1" )
      I_Contact( "DB_Data".F4.Btt_Down_Selected )
      I_Contact( "DB_Data".F5.Btt_Down_Selected )
      I_Contact( "DB_Data".F6.Btt_Down_Selected )
      I_Contact( "DB_Data".F7.Btt_Down_Selected )
      I_Contact( "DB_Data".F8.Btt_Down_Selected )
      I_Contact( "DB_Data".F9.Btt_Down_Selected )
      I_Contact( "DB_Data".F10.Btt_Down_Selected )
      I_Contact( "DB_Data".F11.Btt_Down_Selected )
      I_Contact( "DB_Data".F12.Btt_Down_Selected )
      I_Contact( "DB_Data".F13.Btt_Down_Selected )
      I_Contact( "DB_Data".F14.Btt_Down_Selected )
      I_Contact( "DB_Data".F15.Btt_Down_Selected )
      I_Contact( "DB_Data".F16.Btt_Down_Selected )
      I_Contact( "DB_Data".F17.Btt_Down_Selected )
      I_Contact( "DB_Data".F18.Btt_Down_Selected )
      I_Contact( "DB_Data".F19.Btt_Down_Selected )
      I_Contact( "DB_Data".F20.Btt_Down_Selected )
      P_Trig( "P171" )
      S_Coil( "Q_Door_Open" )
      R_Coil( "Q_Eleveytor_Up" )
      R_Coil( "DB_Data".F3.Btt_Down_Selected )
   END_RUNG
   RUNG wire#w1
      Contact( "DB_Data".F4.Sensor_Correct_Position )
      wire#w4
      Contact( "Q_Eleveytor_Up" )
      Contact( "DB_Data".F4.Btt_Up_Selected )
      P_Trig( "P35" )
      S_Coil( "Q_Door_Open" )
      R_Coil( "Q_Eleveytor_Up" )
      R_Coil( "Q_Eleveytor_Down" )
      R_Coil( "DB_Data".F4.Btt_Up_Selected )
   END_RUNG
   RUNG wire#w4
      Contact( "Q_Eleveytor_Down" )
      Contact( "DB_Data".F4.Btt_Down_Selected )
      P_Trig( "P139" )
      S_Coil( "Q_Door_Open" )
      R_Coil( "Q_Eleveytor_Down" )
      R_Coil( "Q_Eleveytor_Up" )
      R_Coil( "DB_Data".F4.Btt_Down_Selected )
   END_RUNG
   RUNG wire#w4
      Contact( "Q_Eleveytor_Up" )
      Contact( "DB_Data".F4.Btt_Down_Selected )
      Contact( "M_Check1" )
      I_Contact( "DB_Data".F5.Btt_Down_Selected )
      I_Contact( "DB_Data".F6.Btt_Down_Selected )
      I_Contact( "DB_Data".F7.Btt_Down_Selected )
      I_Contact( "DB_Data".F8.Btt_Down_Selected )
      I_Contact( "DB_Data".F9.Btt_Down_Selected )
      I_Contact( "DB_Data".F10.Btt_Down_Selected )
      I_Contact( "DB_Data".F11.Btt_Down_Selected )
      I_Contact( "DB_Data".F12.Btt_Down_Selected )
      I_Contact( "DB_Data".F13.Btt_Down_Selected )
      I_Contact( "DB_Data".F14.Btt_Down_Selected )
      I_Contact( "DB_Data".F15.Btt_Down_Selected )
      I_Contact( "DB_Data".F16.Btt_Down_Selected )
      I_Contact( "DB_Data".F17.Btt_Down_Selected )
      I_Contact( "DB_Data".F18.Btt_Down_Selected )
      I_Contact( "DB_Data".F19.Btt_Down_Selected )
      I_Contact( "DB_Data".F20.Btt_Down_Selected )
      P_Trig( "P172" )
      S_Coil( "Q_Door_Open" )
      R_Coil( "Q_Eleveytor_Up" )
      R_Coil( "DB_Data".F4.Btt_Down_Selected )
   END_RUNG
   RUNG wire#w1
      Contact( "DB_Data".F5.Sensor_Correct_Position )
      wire#w5
      Contact( "Q_Eleveytor_Up" )
      Contact( "DB_Data".F5.Btt_Up_Selected )
      P_Trig( "P140" )
      S_Coil( "Q_Door_Open" )
      R_Coil( "Q_Eleveytor_Up" )
      R_Coil( "Q_Eleveytor_Down" )
      R_Coil( "DB_Data".F5.Btt_Up_Selected )
   END_RUNG
   RUNG wire#w5
      Contact( "Q_Eleveytor_Down" )
      Contact( "DB_Data".F5.Btt_Down_Selected )
      P_Trig( "P141" )
      S_Coil( "Q_Door_Open" )
      R_Coil( "Q_Eleveytor_Down" )
      R_Coil( "Q_Eleveytor_Up" )
      R_Coil( "DB_Data".F5.Btt_Down_Selected )
   END_RUNG
   RUNG wire#w5
      Contact( "Q_Eleveytor_Up" )
      Contact( "DB_Data".F5.Btt_Down_Selected )
      Contact( "M_Check1" )
      I_Contact( "DB_Data".F6.Btt_Down_Selected )
      I_Contact( "DB_Data".F7.Btt_Down_Selected )
      I_Contact( "DB_Data".F8.Btt_Down_Selected )
      I_Contact( "DB_Data".F9.Btt_Down_Selected )
      I_Contact( "DB_Data".F10.Btt_Down_Selected )
      I_Contact( "DB_Data".F11.Btt_Down_Selected )
      I_Contact( "DB_Data".F12.Btt_Down_Selected )
      I_Contact( "DB_Data".F13.Btt_Down_Selected )
      I_Contact( "DB_Data".F14.Btt_Down_Selected )
      I_Contact( "DB_Data".F15.Btt_Down_Selected )
      I_Contact( "DB_Data".F16.Btt_Down_Selected )
      I_Contact( "DB_Data".F17.Btt_Down_Selected )
      I_Contact( "DB_Data".F18.Btt_Down_Selected )
      I_Contact( "DB_Data".F19.Btt_Down_Selected )
      I_Contact( "DB_Data".F20.Btt_Down_Selected )
      P_Trig( "P173" )
      S_Coil( "Q_Door_Open" )
      R_Coil( "Q_Eleveytor_Up" )
      R_Coil( "DB_Data".F5.Btt_Down_Selected )
   END_RUNG
   RUNG wire#w1
      Contact( "DB_Data".F6.Sensor_Correct_Position )
      wire#w6
      Contact( "Q_Eleveytor_Up" )
      Contact( "DB_Data".F6.Btt_Up_Selected )
      P_Trig( "P142" )
      S_Coil( "Q_Door_Open" )
      R_Coil( "Q_Eleveytor_Up" )
      R_Coil( "Q_Eleveytor_Down" )
      R_Coil( "DB_Data".F6.Btt_Up_Selected )
   END_RUNG
   RUNG wire#w6
      Contact( "Q_Eleveytor_Down" )
      Contact( "DB_Data".F6.Btt_Down_Selected )
      P_Trig( "P143" )
      S_Coil( "Q_Door_Open" )
      R_Coil( "Q_Eleveytor_Down" )
      R_Coil( "Q_Eleveytor_Up" )
      R_Coil( "DB_Data".F6.Btt_Down_Selected )
   END_RUNG
   RUNG wire#w6
      Contact( "Q_Eleveytor_Up" )
      Contact( "DB_Data".F6.Btt_Down_Selected )
      Contact( "M_Check1" )
      I_Contact( "DB_Data".F7.Btt_Down_Selected )
      I_Contact( "DB_Data".F8.Btt_Down_Selected )
      I_Contact( "DB_Data".F9.Btt_Down_Selected )
      I_Contact( "DB_Data".F10.Btt_Down_Selected )
      I_Contact( "DB_Data".F11.Btt_Down_Selected )
      I_Contact( "DB_Data".F12.Btt_Down_Selected )
      I_Contact( "DB_Data".F13.Btt_Down_Selected )
      I_Contact( "DB_Data".F14.Btt_Down_Selected )
      I_Contact( "DB_Data".F15.Btt_Down_Selected )
      I_Contact( "DB_Data".F16.Btt_Down_Selected )
      I_Contact( "DB_Data".F17.Btt_Down_Selected )
      I_Contact( "DB_Data".F18.Btt_Down_Selected )
      I_Contact( "DB_Data".F19.Btt_Down_Selected )
      I_Contact( "DB_Data".F20.Btt_Down_Selected )
      P_Trig( "P174" )
      S_Coil( "Q_Door_Open" )
      R_Coil( "Q_Eleveytor_Up" )
      R_Coil( "DB_Data".F6.Btt_Down_Selected )
   END_RUNG
   RUNG wire#w1
      Contact( "DB_Data".F7.Sensor_Correct_Position )
      wire#w7
      Contact( "Q_Eleveytor_Up" )
      Contact( "DB_Data".F7.Btt_Up_Selected )
      P_Trig( "P144" )
      S_Coil( "Q_Door_Open" )
      R_Coil( "Q_Eleveytor_Up" )
      R_Coil( "Q_Eleveytor_Down" )
      R_Coil( "DB_Data".F7.Btt_Up_Selected )
   END_RUNG
   RUNG wire#w7
      Contact( "Q_Eleveytor_Down" )
      Contact( "DB_Data".F7.Btt_Down_Selected )
      P_Trig( "P145" )
      S_Coil( "Q_Door_Open" )
      R_Coil( "Q_Eleveytor_Down" )
      R_Coil( "Q_Eleveytor_Up" )
      R_Coil( "DB_Data".F7.Btt_Down_Selected )
   END_RUNG
   RUNG wire#w7
      Contact( "Q_Eleveytor_Up" )
      Contact( "DB_Data".F7.Btt_Down_Selected )
      Contact( "M_Check1" )
      I_Contact( "DB_Data".F8.Btt_Down_Selected )
      I_Contact( "DB_Data".F9.Btt_Down_Selected )
      I_Contact( "DB_Data".F10.Btt_Down_Selected )
      I_Contact( "DB_Data".F11.Btt_Down_Selected )
      I_Contact( "DB_Data".F12.Btt_Down_Selected )
      I_Contact( "DB_Data".F13.Btt_Down_Selected )
      I_Contact( "DB_Data".F14.Btt_Down_Selected )
      I_Contact( "DB_Data".F15.Btt_Down_Selected )
      I_Contact( "DB_Data".F16.Btt_Down_Selected )
      I_Contact( "DB_Data".F17.Btt_Down_Selected )
      I_Contact( "DB_Data".F18.Btt_Down_Selected )
      I_Contact( "DB_Data".F19.Btt_Down_Selected )
      I_Contact( "DB_Data".F20.Btt_Down_Selected )
      P_Trig( "P175" )
      S_Coil( "Q_Door_Open" )
      R_Coil( "Q_Eleveytor_Up" )
      R_Coil( "DB_Data".F7.Btt_Down_Selected )
   END_RUNG
   RUNG wire#w1
      Contact( "DB_Data".F8.Sensor_Correct_Position )
      wire#w8
      Contact( "Q_Eleveytor_Up" )
      Contact( "DB_Data".F8.Btt_Up_Selected )
      P_Trig( "P146" )
      S_Coil( "Q_Door_Open" )
      R_Coil( "Q_Eleveytor_Up" )
      R_Coil( "Q_Eleveytor_Down" )
      R_Coil( "DB_Data".F8.Btt_Up_Selected )
   END_RUNG
   RUNG wire#w8
      Contact( "Q_Eleveytor_Down" )
      Contact( "DB_Data".F8.Btt_Down_Selected )
      P_Trig( "P147" )
      S_Coil( "Q_Door_Open" )
      R_Coil( "Q_Eleveytor_Down" )
      R_Coil( "Q_Eleveytor_Up" )
      R_Coil( "DB_Data".F8.Btt_Down_Selected )
   END_RUNG
   RUNG wire#w8
      Contact( "Q_Eleveytor_Up" )
      Contact( "DB_Data".F8.Btt_Down_Selected )
      Contact( "M_Check1" )
      I_Contact( "DB_Data".F9.Btt_Down_Selected )
      I_Contact( "DB_Data".F10.Btt_Down_Selected )
      I_Contact( "DB_Data".F11.Btt_Down_Selected )
      I_Contact( "DB_Data".F12.Btt_Down_Selected )
      I_Contact( "DB_Data".F13.Btt_Down_Selected )
      I_Contact( "DB_Data".F14.Btt_Down_Selected )
      I_Contact( "DB_Data".F15.Btt_Down_Selected )
      I_Contact( "DB_Data".F16.Btt_Down_Selected )
      I_Contact( "DB_Data".F17.Btt_Down_Selected )
      I_Contact( "DB_Data".F18.Btt_Down_Selected )
      I_Contact( "DB_Data".F19.Btt_Down_Selected )
      I_Contact( "DB_Data".F20.Btt_Down_Selected )
      P_Trig( "P176" )
      S_Coil( "Q_Door_Open" )
      R_Coil( "Q_Eleveytor_Up" )
      R_Coil( "DB_Data".F8.Btt_Down_Selected )
   END_RUNG
   RUNG wire#w1
      Contact( "DB_Data".F9.Sensor_Correct_Position )
      wire#w9
      Contact( "Q_Eleveytor_Up" )
      Contact( "DB_Data".F9.Btt_Up_Selected )
      P_Trig( "P148" )
      S_Coil( "Q_Door_Open" )
      R_Coil( "Q_Eleveytor_Up" )
      R_Coil( "Q_Eleveytor_Down" )
      R_Coil( "DB_Data".F9.Btt_Up_Selected )
   END_RUNG
   RUNG wire#w9
      Contact( "Q_Eleveytor_Down" )
      Contact( "DB_Data".F9.Btt_Down_Selected )
      P_Trig( "P149" )
      S_Coil( "Q_Door_Open" )
      R_Coil( "Q_Eleveytor_Down" )
      R_Coil( "Q_Eleveytor_Up" )
      R_Coil( "DB_Data".F9.Btt_Down_Selected )
   END_RUNG
   RUNG wire#w9
      Contact( "Q_Eleveytor_Up" )
      Contact( "DB_Data".F9.Btt_Down_Selected )
      Contact( "M_Check1" )
      I_Contact( "DB_Data".F10.Btt_Down_Selected )
      I_Contact( "DB_Data".F11.Btt_Down_Selected )
      I_Contact( "DB_Data".F12.Btt_Down_Selected )
      I_Contact( "DB_Data".F13.Btt_Down_Selected )
      I_Contact( "DB_Data".F14.Btt_Down_Selected )
      I_Contact( "DB_Data".F15.Btt_Down_Selected )
      I_Contact( "DB_Data".F16.Btt_Down_Selected )
      I_Contact( "DB_Data".F17.Btt_Down_Selected )
      I_Contact( "DB_Data".F18.Btt_Down_Selected )
      I_Contact( "DB_Data".F19.Btt_Down_Selected )
      I_Contact( "DB_Data".F20.Btt_Down_Selected )
      P_Trig( "P177" )
      S_Coil( "Q_Door_Open" )
      R_Coil( "Q_Eleveytor_Up" )
      R_Coil( "DB_Data".F9.Btt_Down_Selected )
   END_RUNG
   RUNG wire#w1
      Contact( "DB_Data".F10.Sensor_Correct_Position )
      wire#w10
      Contact( "Q_Eleveytor_Up" )
      Contact( "DB_Data".F10.Btt_Up_Selected )
      P_Trig( "P150" )
      S_Coil( "Q_Door_Open" )
      R_Coil( "Q_Eleveytor_Up" )
      R_Coil( "Q_Eleveytor_Down" )
      R_Coil( "DB_Data".F10.Btt_Up_Selected )
   END_RUNG
   RUNG wire#w10
      Contact( "Q_Eleveytor_Down" )
      Contact( "DB_Data".F10.Btt_Down_Selected )
      P_Trig( "P48" )
      S_Coil( "Q_Door_Open" )
      R_Coil( "Q_Eleveytor_Down" )
      R_Coil( "Q_Eleveytor_Up" )
      R_Coil( "DB_Data".F10.Btt_Down_Selected )
   END_RUNG
   RUNG wire#w10
      Contact( "Q_Eleveytor_Up" )
      Contact( "DB_Data".F10.Btt_Down_Selected )
      Contact( "M_Check1" )
      I_Contact( "DB_Data".F11.Btt_Down_Selected )
      I_Contact( "DB_Data".F12.Btt_Down_Selected )
      I_Contact( "DB_Data".F13.Btt_Down_Selected )
      I_Contact( "DB_Data".F14.Btt_Down_Selected )
      I_Contact( "DB_Data".F15.Btt_Down_Selected )
      I_Contact( "DB_Data".F16.Btt_Down_Selected )
      I_Contact( "DB_Data".F17.Btt_Down_Selected )
      I_Contact( "DB_Data".F18.Btt_Down_Selected )
      I_Contact( "DB_Data".F19.Btt_Down_Selected )
      I_Contact( "DB_Data".F20.Btt_Down_Selected )
      P_Trig( "P178" )
      S_Coil( "Q_Door_Open" )
      R_Coil( "Q_Eleveytor_Up" )
      R_Coil( "DB_Data".F10.Btt_Down_Selected )
   END_RUNG
   RUNG wire#w1
      Contact( "DB_Data".F11.Sensor_Correct_Position )
      wire#w11
      Contact( "Q_Eleveytor_Up" )
      Contact( "DB_Data".F11.Btt_Up_Selected )
      P_Trig( "P151" )
      S_Coil( "Q_Door_Open" )
      R_Coil( "Q_Eleveytor_Up" )
      R_Coil( "Q_Eleveytor_Down" )
      R_Coil( "DB_Data".F11.Btt_Up_Selected )
   END_RUNG
   RUNG wire#w11
      Contact( "Q_Eleveytor_Down" )
      Contact( "DB_Data".F11.Btt_Down_Selected )
      P_Trig( "P152" )
      S_Coil( "Q_Door_Open" )
      R_Coil( "Q_Eleveytor_Down" )
      R_Coil( "Q_Eleveytor_Up" )
      R_Coil( "DB_Data".F11.Btt_Down_Selected )
   END_RUNG
   RUNG wire#w11
      Contact( "Q_Eleveytor_Up" )
      Contact( "DB_Data".F11.Btt_Down_Selected )
      Contact( "M_Check1" )
      I_Contact( "DB_Data".F12.Btt_Down_Selected )
      I_Contact( "DB_Data".F13.Btt_Down_Selected )
      I_Contact( "DB_Data".F14.Btt_Down_Selected )
      I_Contact( "DB_Data".F15.Btt_Down_Selected )
      I_Contact( "DB_Data".F16.Btt_Down_Selected )
      I_Contact( "DB_Data".F17.Btt_Down_Selected )
      I_Contact( "DB_Data".F18.Btt_Down_Selected )
      I_Contact( "DB_Data".F19.Btt_Down_Selected )
      I_Contact( "DB_Data".F20.Btt_Down_Selected )
      P_Trig( "P179" )
      S_Coil( "Q_Door_Open" )
      R_Coil( "Q_Eleveytor_Up" )
      R_Coil( "DB_Data".F11.Btt_Down_Selected )
   END_RUNG
   RUNG wire#w1
      Contact( "DB_Data".F12.Sensor_Correct_Position )
      wire#w12
      Contact( "Q_Eleveytor_Up" )
      Contact( "DB_Data".F12.Btt_Up_Selected )
      P_Trig( "P153" )
      S_Coil( "Q_Door_Open" )
      R_Coil( "Q_Eleveytor_Up" )
      R_Coil( "Q_Eleveytor_Down" )
      R_Coil( "DB_Data".F12.Btt_Up_Selected )
   END_RUNG
   RUNG wire#w12
      Contact( "Q_Eleveytor_Down" )
      Contact( "DB_Data".F12.Btt_Down_Selected )
      P_Trig( "P154" )
      S_Coil( "Q_Door_Open" )
      R_Coil( "Q_Eleveytor_Down" )
      R_Coil( "Q_Eleveytor_Up" )
      R_Coil( "DB_Data".F12.Btt_Down_Selected )
   END_RUNG
   RUNG wire#w12
      Contact( "Q_Eleveytor_Up" )
      Contact( "DB_Data".F12.Btt_Down_Selected )
      Contact( "M_Check1" )
      I_Contact( "DB_Data".F13.Btt_Down_Selected )
      I_Contact( "DB_Data".F14.Btt_Down_Selected )
      I_Contact( "DB_Data".F15.Btt_Down_Selected )
      I_Contact( "DB_Data".F16.Btt_Down_Selected )
      I_Contact( "DB_Data".F17.Btt_Down_Selected )
      I_Contact( "DB_Data".F18.Btt_Down_Selected )
      I_Contact( "DB_Data".F19.Btt_Down_Selected )
      I_Contact( "DB_Data".F20.Btt_Down_Selected )
      P_Trig( "P180" )
      S_Coil( "Q_Door_Open" )
      R_Coil( "Q_Eleveytor_Up" )
      R_Coil( "DB_Data".F12.Btt_Down_Selected )
   END_RUNG
   RUNG wire#w1
      Contact( "DB_Data".F13.Sensor_Correct_Position )
      wire#w13
      Contact( "Q_Eleveytor_Up" )
      Contact( "DB_Data".F13.Btt_Up_Selected )
      P_Trig( "P155" )
      S_Coil( "Q_Door_Open" )
      R_Coil( "Q_Eleveytor_Up" )
      R_Coil( "Q_Eleveytor_Down" )
      R_Coil( "DB_Data".F13.Btt_Up_Selected )
   END_RUNG
   RUNG wire#w13
      Contact( "Q_Eleveytor_Down" )
      Contact( "DB_Data".F13.Btt_Down_Selected )
      P_Trig( "P156" )
      S_Coil( "Q_Door_Open" )
      R_Coil( "Q_Eleveytor_Down" )
      R_Coil( "Q_Eleveytor_Up" )
      R_Coil( "DB_Data".F13.Btt_Down_Selected )
   END_RUNG
   RUNG wire#w13
      Contact( "Q_Eleveytor_Up" )
      Contact( "DB_Data".F13.Btt_Down_Selected )
      Contact( "M_Check1" )
      I_Contact( "DB_Data".F14.Btt_Down_Selected )
      I_Contact( "DB_Data".F15.Btt_Down_Selected )
      I_Contact( "DB_Data".F16.Btt_Down_Selected )
      I_Contact( "DB_Data".F17.Btt_Down_Selected )
      I_Contact( "DB_Data".F18.Btt_Down_Selected )
      I_Contact( "DB_Data".F19.Btt_Down_Selected )
      I_Contact( "DB_Data".F20.Btt_Down_Selected )
      P_Trig( "P181" )
      S_Coil( "Q_Door_Open" )
      R_Coil( "Q_Eleveytor_Up" )
      R_Coil( "DB_Data".F13.Btt_Down_Selected )
   END_RUNG
   RUNG wire#w1
      Contact( "DB_Data".F14.Sensor_Correct_Position )
      wire#w14
      Contact( "Q_Eleveytor_Up" )
      Contact( "DB_Data".F14.Btt_Up_Selected )
      P_Trig( "P157" )
      S_Coil( "Q_Door_Open" )
      R_Coil( "Q_Eleveytor_Up" )
      R_Coil( "Q_Eleveytor_Down" )
      R_Coil( "DB_Data".F14.Btt_Up_Selected )
   END_RUNG
   RUNG wire#w14
      Contact( "Q_Eleveytor_Down" )
      Contact( "DB_Data".F14.Btt_Down_Selected )
      P_Trig( "P158" )
      S_Coil( "Q_Door_Open" )
      R_Coil( "Q_Eleveytor_Down" )
      R_Coil( "Q_Eleveytor_Up" )
      R_Coil( "DB_Data".F14.Btt_Down_Selected )
   END_RUNG
   RUNG wire#w14
      Contact( "Q_Eleveytor_Up" )
      Contact( "DB_Data".F14.Btt_Down_Selected )
      Contact( "M_Check1" )
      I_Contact( "DB_Data".F15.Btt_Down_Selected )
      I_Contact( "DB_Data".F16.Btt_Down_Selected )
      I_Contact( "DB_Data".F17.Btt_Down_Selected )
      I_Contact( "DB_Data".F18.Btt_Down_Selected )
      I_Contact( "DB_Data".F19.Btt_Down_Selected )
      I_Contact( "DB_Data".F20.Btt_Down_Selected )
      P_Trig( "P182" )
      S_Coil( "Q_Door_Open" )
      R_Coil( "Q_Eleveytor_Up" )
      R_Coil( "DB_Data".F14.Btt_Down_Selected )
   END_RUNG
   RUNG wire#w1
      Contact( "DB_Data".F15.Sensor_Correct_Position )
      wire#w15
      Contact( "Q_Eleveytor_Up" )
      Contact( "DB_Data".F15.Btt_Up_Selected )
      P_Trig( "P159" )
      S_Coil( "Q_Door_Open" )
      R_Coil( "Q_Eleveytor_Up" )
      R_Coil( "Q_Eleveytor_Down" )
      R_Coil( "DB_Data".F15.Btt_Up_Selected )
   END_RUNG
   RUNG wire#w15
      Contact( "Q_Eleveytor_Down" )
      Contact( "DB_Data".F15.Btt_Down_Selected )
      P_Trig( "P160" )
      S_Coil( "Q_Door_Open" )
      R_Coil( "Q_Eleveytor_Down" )
      R_Coil( "Q_Eleveytor_Up" )
      R_Coil( "DB_Data".F15.Btt_Down_Selected )
   END_RUNG
   RUNG wire#w15
      Contact( "Q_Eleveytor_Up" )
      Contact( "DB_Data".F15.Btt_Down_Selected )
      Contact( "M_Check1" )
      I_Contact( "DB_Data".F16.Btt_Down_Selected )
      I_Contact( "DB_Data".F17.Btt_Down_Selected )
      I_Contact( "DB_Data".F18.Btt_Down_Selected )
      I_Contact( "DB_Data".F19.Btt_Down_Selected )
      I_Contact( "DB_Data".F20.Btt_Down_Selected )
      P_Trig( "P183" )
      S_Coil( "Q_Door_Open" )
      R_Coil( "Q_Eleveytor_Up" )
      R_Coil( "DB_Data".F15.Btt_Down_Selected )
   END_RUNG
   RUNG wire#w1
      Contact( "DB_Data".F16.Sensor_Correct_Position )
      wire#w16
      Contact( "Q_Eleveytor_Up" )
      Contact( "DB_Data".F16.Btt_Up_Selected )
      P_Trig( "P161" )
      S_Coil( "Q_Door_Open" )
      R_Coil( "Q_Eleveytor_Up" )
      R_Coil( "Q_Eleveytor_Down" )
      R_Coil( "DB_Data".F16.Btt_Up_Selected )
   END_RUNG
   RUNG wire#w16
      Contact( "Q_Eleveytor_Down" )
      Contact( "DB_Data".F16.Btt_Down_Selected )
      P_Trig( "P162" )
      S_Coil( "Q_Door_Open" )
      R_Coil( "Q_Eleveytor_Down" )
      R_Coil( "Q_Eleveytor_Up" )
      R_Coil( "DB_Data".F16.Btt_Down_Selected )
   END_RUNG
   RUNG wire#w16
      Contact( "Q_Eleveytor_Up" )
      Contact( "DB_Data".F16.Btt_Down_Selected )
      Contact( "M_Check1" )
      I_Contact( "DB_Data".F17.Btt_Down_Selected )
      I_Contact( "DB_Data".F18.Btt_Down_Selected )
      I_Contact( "DB_Data".F19.Btt_Down_Selected )
      I_Contact( "DB_Data".F20.Btt_Down_Selected )
      P_Trig( "P183" )
      S_Coil( "Q_Door_Open" )
      R_Coil( "Q_Eleveytor_Up" )
      R_Coil( "DB_Data".F16.Btt_Down_Selected )
   END_RUNG
   RUNG wire#w1
      Contact( "DB_Data".F17.Sensor_Correct_Position )
      wire#w17
      Contact( "Q_Eleveytor_Up" )
      Contact( "DB_Data".F17.Btt_Up_Selected )
      P_Trig( "P163" )
      S_Coil( "Q_Door_Open" )
      R_Coil( "Q_Eleveytor_Up" )
      R_Coil( "Q_Eleveytor_Down" )
      R_Coil( "DB_Data".F17.Btt_Up_Selected )
   END_RUNG
   RUNG wire#w17
      Contact( "Q_Eleveytor_Down" )
      Contact( "DB_Data".F17.Btt_Down_Selected )
      P_Trig( "P164" )
      S_Coil( "Q_Door_Open" )
      R_Coil( "Q_Eleveytor_Down" )
      R_Coil( "Q_Eleveytor_Up" )
      R_Coil( "DB_Data".F17.Btt_Down_Selected )
   END_RUNG
   RUNG wire#w17
      Contact( "Q_Eleveytor_Up" )
      Contact( "DB_Data".F17.Btt_Down_Selected )
      Contact( "M_Check1" )
      I_Contact( "DB_Data".F18.Btt_Down_Selected )
      I_Contact( "DB_Data".F19.Btt_Down_Selected )
      I_Contact( "DB_Data".F20.Btt_Down_Selected )
      P_Trig( "P184" )
      S_Coil( "Q_Door_Open" )
      R_Coil( "Q_Eleveytor_Up" )
      R_Coil( "DB_Data".F17.Btt_Down_Selected )
   END_RUNG
   RUNG wire#w1
      Contact( "DB_Data".F18.Sensor_Correct_Position )
      wire#w18
      Contact( "Q_Eleveytor_Up" )
      Contact( "DB_Data".F18.Btt_Up_Selected )
      P_Trig( "P165" )
      S_Coil( "Q_Door_Open" )
      R_Coil( "Q_Eleveytor_Up" )
      R_Coil( "Q_Eleveytor_Down" )
      R_Coil( "DB_Data".F18.Btt_Up_Selected )
   END_RUNG
   RUNG wire#w18
      Contact( "Q_Eleveytor_Down" )
      Contact( "DB_Data".F18.Btt_Down_Selected )
      P_Trig( "P166" )
      S_Coil( "Q_Door_Open" )
      R_Coil( "Q_Eleveytor_Down" )
      R_Coil( "Q_Eleveytor_Up" )
      R_Coil( "DB_Data".F18.Btt_Down_Selected )
   END_RUNG
   RUNG wire#w18
      Contact( "Q_Eleveytor_Up" )
      Contact( "DB_Data".F18.Btt_Down_Selected )
      Contact( "M_Check1" )
      I_Contact( "DB_Data".F19.Btt_Down_Selected )
      I_Contact( "DB_Data".F20.Btt_Down_Selected )
      P_Trig( "P185" )
      S_Coil( "Q_Door_Open" )
      R_Coil( "Q_Eleveytor_Up" )
      R_Coil( "DB_Data".F18.Btt_Down_Selected )
   END_RUNG
   RUNG wire#w1
      Contact( "DB_Data".F19.Sensor_Correct_Position )
      wire#w19
      Contact( "Q_Eleveytor_Up" )
      Contact( "DB_Data".F19.Btt_Up_Selected )
      P_Trig( "P167" )
      S_Coil( "Q_Door_Open" )
      R_Coil( "Q_Eleveytor_Up" )
      R_Coil( "Q_Eleveytor_Down" )
      R_Coil( "DB_Data".F19.Btt_Up_Selected )
   END_RUNG
   RUNG wire#w19
      Contact( "Q_Eleveytor_Down" )
      Contact( "DB_Data".F19.Btt_Down_Selected )
      P_Trig( "P168" )
      S_Coil( "Q_Door_Open" )
      R_Coil( "Q_Eleveytor_Down" )
      R_Coil( "Q_Eleveytor_Up" )
      R_Coil( "DB_Data".F19.Btt_Down_Selected )
   END_RUNG
   RUNG wire#w19
      Contact( "Q_Eleveytor_Up" )
      Contact( "DB_Data".F19.Btt_Down_Selected )
      Contact( "M_Check1" )
      I_Contact( "DB_Data".F20.Btt_Down_Selected )
      P_Trig( "P186" )
      S_Coil( "Q_Door_Open" )
      R_Coil( "Q_Eleveytor_Up" )
      R_Coil( "DB_Data".F19.Btt_Down_Selected )
   END_RUNG
   RUNG wire#w1
      Contact( "DB_Data".F20.Sensor_Correct_Position )
      Contact( "Q_Eleveytor_Up" )
      Contact( "DB_Data".F20.Btt_Down_Selected )
      P_Trig( "P169" )
      S_Coil( "Q_Door_Open" )
      R_Coil( "Q_Eleveytor_Up" )
      R_Coil( "DB_Data".F20.Btt_Down_Selected )
   END_RUNG
   // the same network as SCL:
   #_w1 := NOT "AlwaysFALSE" AND "DB_Data".F1.Sensor_Correct_Position AND "Q_Eleveytor_Down" AND "DB_Data".F1.Btt_Up_Selected;
   #_w2 := #_w1 AND NOT "P30";   // rising edge
   "P30" := #_w1;
   IF #_w2 THEN
       "Q_Door_Open" := TRUE;
       "Q_Eleveytor_Down" := FALSE;
       "DB_Data".F1.Btt_Up_Selected := FALSE;
   END_IF;
   #_w3 := NOT "AlwaysFALSE" AND "DB_Data".F2.Sensor_Correct_Position;
   #_w4 := #_w3 AND "Q_Eleveytor_Up" AND "DB_Data".F2.Btt_Up_Selected;
   #_w5 := #_w4 AND NOT "P31";   // rising edge
   "P31" := #_w4;
   IF #_w5 THEN
       "Q_Door_Open" := TRUE;
       "Q_Eleveytor_Up" := FALSE;
       "Q_Eleveytor_Down" := FALSE;
       "DB_Data".F2.Btt_Up_Selected := FALSE;
   END_IF;
   #_w6 := #_w3 AND "Q_Eleveytor_Down" AND "DB_Data".F2.Btt_Down_Selected;
   #_w7 := #_w6 AND NOT "P32";   // rising edge
   "P32" := #_w6;
   IF #_w7 THEN
       "Q_Door_Open" := TRUE;
       "Q_Eleveytor_Down" := FALSE;
       "Q_Eleveytor_Up" := FALSE;
       "DB_Data".F2.Btt_Down_Selected := FALSE;
   END_IF;
   #_w8 := #_w3 AND "Q_Eleveytor_Up" AND "DB_Data".F2.Btt_Down_Selected AND "M_Check1" AND NOT "DB_Data".F3.Btt_Down_Selected AND NOT "DB_Data".F4.Btt_Down_Selected AND NOT "DB_Data".F5.Btt_Down_Selected AND NOT "DB_Data".F6.Btt_Down_Selected AND NOT "DB_Data".F7.Btt_Down_Selected AND NOT "DB_Data".F8.Btt_Down_Selected AND NOT "DB_Data".F9.Btt_Down_Selected AND NOT "DB_Data".F10.Btt_Down_Selected AND NOT "DB_Data".F11.Btt_Down_Selected AND NOT "DB_Data".F12.Btt_Down_Selected AND NOT "DB_Data".F13.Btt_Down_Selected AND NOT "DB_Data".F14.Btt_Down_Selected AND NOT "DB_Data".F15.Btt_Down_Selected AND NOT "DB_Data".F16.Btt_Down_Selected AND NOT "DB_Data".F17.Btt_Down_Selected AND NOT "DB_Data".F18.Btt_Down_Selected AND NOT "DB_Data".F19.Btt_Down_Selected AND NOT "DB_Data".F20.Btt_Down_Selected;
   #_w9 := #_w8 AND NOT "P170";   // rising edge
   "P170" := #_w8;
   IF #_w9 THEN
       "Q_Door_Open" := TRUE;
       "Q_Eleveytor_Up" := FALSE;
       "DB_Data".F2.Btt_Down_Selected := FALSE;
   END_IF;
   #_w10 := NOT "AlwaysFALSE" AND "DB_Data".F3.Sensor_Correct_Position;
   #_w11 := #_w10 AND "Q_Eleveytor_Up" AND "DB_Data".F3.Btt_Up_Selected;
   #_w12 := #_w11 AND NOT "P33";   // rising edge
   "P33" := #_w11;
   IF #_w12 THEN
       "Q_Door_Open" := TRUE;
       "Q_Eleveytor_Up" := FALSE;
       "Q_Eleveytor_Down" := FALSE;
       "DB_Data".F3.Btt_Up_Selected := FALSE;
   END_IF;
   #_w13 := #_w10 AND "Q_Eleveytor_Down" AND "DB_Data".F3.Btt_Down_Selected;
   #_w14 := #_w13 AND NOT "P34";   // rising edge
   "P34" := #_w13;
   IF #_w14 THEN
       "Q_Door_Open" := TRUE;
       "Q_Eleveytor_Down" := FALSE;
       "Q_Eleveytor_Up" := FALSE;
       "DB_Data".F3.Btt_Down_Selected := FALSE;
   END_IF;
   #_w15 := #_w10 AND "Q_Eleveytor_Up" AND "DB_Data".F3.Btt_Down_Selected AND "M_Check1" AND NOT "DB_Data".F4.Btt_Down_Selected AND NOT "DB_Data".F5.Btt_Down_Selected AND NOT "DB_Data".F6.Btt_Down_Selected AND NOT "DB_Data".F7.Btt_Down_Selected AND NOT "DB_Data".F8.Btt_Down_Selected AND NOT "DB_Data".F9.Btt_Down_Selected AND NOT "DB_Data".F10.Btt_Down_Selected AND NOT "DB_Data".F11.Btt_Down_Selected AND NOT "DB_Data".F12.Btt_Down_Selected AND NOT "DB_Data".F13.Btt_Down_Selected AND NOT "DB_Data".F14.Btt_Down_Selected AND NOT "DB_Data".F15.Btt_Down_Selected AND NOT "DB_Data".F16.Btt_Down_Selected AND NOT "DB_Data".F17.Btt_Down_Selected AND NOT "DB_Data".F18.Btt_Down_Selected AND NOT "DB_Data".F19.Btt_Down_Selected AND NOT "DB_Data".F20.Btt_Down_Selected;
   #_w16 := #_w15 AND NOT "P171";   // rising edge
   "P171" := #_w15;
   IF #_w16 THEN
       "Q_Door_Open" := TRUE;
       "Q_Eleveytor_Up" := FALSE;
       "DB_Data".F3.Btt_Down_Selected := FALSE;
   END_IF;
   #_w17 := NOT "AlwaysFALSE" AND "DB_Data".F4.Sensor_Correct_Position;
   #_w18 := #_w17 AND "Q_Eleveytor_Up" AND "DB_Data".F4.Btt_Up_Selected;
   #_w19 := #_w18 AND NOT "P35";   // rising edge
   "P35" := #_w18;
   IF #_w19 THEN
       "Q_Door_Open" := TRUE;
       "Q_Eleveytor_Up" := FALSE;
       "Q_Eleveytor_Down" := FALSE;
       "DB_Data".F4.Btt_Up_Selected := FALSE;
   END_IF;
   #_w20 := #_w17 AND "Q_Eleveytor_Down" AND "DB_Data".F4.Btt_Down_Selected;
   #_w21 := #_w20 AND NOT "P139";   // rising edge
   "P139" := #_w20;
   IF #_w21 THEN
       "Q_Door_Open" := TRUE;
       "Q_Eleveytor_Down" := FALSE;
       "Q_Eleveytor_Up" := FALSE;
       "DB_Data".F4.Btt_Down_Selected := FALSE;
   END_IF;
   #_w22 := #_w17 AND "Q_Eleveytor_Up" AND "DB_Data".F4.Btt_Down_Selected AND "M_Check1" AND NOT "DB_Data".F5.Btt_Down_Selected AND NOT "DB_Data".F6.Btt_Down_Selected AND NOT "DB_Data".F7.Btt_Down_Selected AND NOT "DB_Data".F8.Btt_Down_Selected AND NOT "DB_Data".F9.Btt_Down_Selected AND NOT "DB_Data".F10.Btt_Down_Selected AND NOT "DB_Data".F11.Btt_Down_Selected AND NOT "DB_Data".F12.Btt_Down_Selected AND NOT "DB_Data".F13.Btt_Down_Selected AND NOT "DB_Data".F14.Btt_Down_Selected AND NOT "DB_Data".F15.Btt_Down_Selected AND NOT "DB_Data".F16.Btt_Down_Selected AND NOT "DB_Data".F17.Btt_Down_Selected AND NOT "DB_Data".F18.Btt_Down_Selected AND NOT "DB_Data".F19.Btt_Down_Selected AND NOT "DB_Data".F20.Btt_Down_Selected;
   #_w23 := #_w22 AND NOT "P172";   // rising edge
   "P172" := #_w22;
   IF #_w23 THEN
       "Q_Door_Open" := TRUE;
       "Q_Eleveytor_Up" := FALSE;
       "DB_Data".F4.Btt_Down_Selected := FALSE;
   END_IF;
   #_w24 := NOT "AlwaysFALSE" AND "DB_Data".F5.Sensor_Correct_Position;
   #_w25 := #_w24 AND "Q_Eleveytor_Up" AND "DB_Data".F5.Btt_Up_Selected;
   #_w26 := #_w25 AND NOT "P140";   // rising edge
   "P140" := #_w25;
   IF #_w26 THEN
       "Q_Door_Open" := TRUE;
       "Q_Eleveytor_Up" := FALSE;
       "Q_Eleveytor_Down" := FALSE;
       "DB_Data".F5.Btt_Up_Selected := FALSE;
   END_IF;
   #_w27 := #_w24 AND "Q_Eleveytor_Down" AND "DB_Data".F5.Btt_Down_Selected;
   #_w28 := #_w27 AND NOT "P141";   // rising edge
   "P141" := #_w27;
   IF #_w28 THEN
       "Q_Door_Open" := TRUE;
       "Q_Eleveytor_Down" := FALSE;
       "Q_Eleveytor_Up" := FALSE;
       "DB_Data".F5.Btt_Down_Selected := FALSE;
   END_IF;
   #_w29 := #_w24 AND "Q_Eleveytor_Up" AND "DB_Data".F5.Btt_Down_Selected AND "M_Check1" AND NOT "DB_Data".F6.Btt_Down_Selected AND NOT "DB_Data".F7.Btt_Down_Selected AND NOT "DB_Data".F8.Btt_Down_Selected AND NOT "DB_Data".F9.Btt_Down_Selected AND NOT "DB_Data".F10.Btt_Down_Selected AND NOT "DB_Data".F11.Btt_Down_Selected AND NOT "DB_Data".F12.Btt_Down_Selected AND NOT "DB_Data".F13.Btt_Down_Selected AND NOT "DB_Data".F14.Btt_Down_Selected AND NOT "DB_Data".F15.Btt_Down_Selected AND NOT "DB_Data".F16.Btt_Down_Selected AND NOT "DB_Data".F17.Btt_Down_Selected AND NOT "DB_Data".F18.Btt_Down_Selected AND NOT "DB_Data".F19.Btt_Down_Selected AND NOT "DB_Data".F20.Btt_Down_Selected;
   #_w30 := #_w29 AND NOT "P173";   // rising edge
   "P173" := #_w29;
   IF #_w30 THEN
       "Q_Door_Open" := TRUE;
       "Q_Eleveytor_Up" := FALSE;
       "DB_Data".F5.Btt_Down_Selected := FALSE;
   END_IF;
   #_w31 := NOT "AlwaysFALSE" AND "DB_Data".F6.Sensor_Correct_Position;
   #_w32 := #_w31 AND "Q_Eleveytor_Up" AND "DB_Data".F6.Btt_Up_Selected;
   #_w33 := #_w32 AND NOT "P142";   // rising edge
   "P142" := #_w32;
   IF #_w33 THEN
       "Q_Door_Open" := TRUE;
       "Q_Eleveytor_Up" := FALSE;
       "Q_Eleveytor_Down" := FALSE;
       "DB_Data".F6.Btt_Up_Selected := FALSE;
   END_IF;
   #_w34 := #_w31 AND "Q_Eleveytor_Down" AND "DB_Data".F6.Btt_Down_Selected;
   #_w35 := #_w34 AND NOT "P143";   // rising edge
   "P143" := #_w34;
   IF #_w35 THEN
       "Q_Door_Open" := TRUE;
       "Q_Eleveytor_Down" := FALSE;
       "Q_Eleveytor_Up" := FALSE;
       "DB_Data".F6.Btt_Down_Selected := FALSE;
   END_IF;
   #_w36 := #_w31 AND "Q_Eleveytor_Up" AND "DB_Data".F6.Btt_Down_Selected AND "M_Check1" AND NOT "DB_Data".F7.Btt_Down_Selected AND NOT "DB_Data".F8.Btt_Down_Selected AND NOT "DB_Data".F9.Btt_Down_Selected AND NOT "DB_Data".F10.Btt_Down_Selected AND NOT "DB_Data".F11.Btt_Down_Selected AND NOT "DB_Data".F12.Btt_Down_Selected AND NOT "DB_Data".F13.Btt_Down_Selected AND NOT "DB_Data".F14.Btt_Down_Selected AND NOT "DB_Data".F15.Btt_Down_Selected AND NOT "DB_Data".F16.Btt_Down_Selected AND NOT "DB_Data".F17.Btt_Down_Selected AND NOT "DB_Data".F18.Btt_Down_Selected AND NOT "DB_Data".F19.Btt_Down_Selected AND NOT "DB_Data".F20.Btt_Down_Selected;
   #_w37 := #_w36 AND NOT "P174";   // rising edge
   "P174" := #_w36;
   IF #_w37 THEN
       "Q_Door_Open" := TRUE;
       "Q_Eleveytor_Up" := FALSE;
       "DB_Data".F6.Btt_Down_Selected := FALSE;
   END_IF;
   #_w38 := NOT "AlwaysFALSE" AND "DB_Data".F7.Sensor_Correct_Position;
   #_w39 := #_w38 AND "Q_Eleveytor_Up" AND "DB_Data".F7.Btt_Up_Selected;
   #_w40 := #_w39 AND NOT "P144";   // rising edge
   "P144" := #_w39;
   IF #_w40 THEN
       "Q_Door_Open" := TRUE;
       "Q_Eleveytor_Up" := FALSE;
       "Q_Eleveytor_Down" := FALSE;
       "DB_Data".F7.Btt_Up_Selected := FALSE;
   END_IF;
   #_w41 := #_w38 AND "Q_Eleveytor_Down" AND "DB_Data".F7.Btt_Down_Selected;
   #_w42 := #_w41 AND NOT "P145";   // rising edge
   "P145" := #_w41;
   IF #_w42 THEN
       "Q_Door_Open" := TRUE;
       "Q_Eleveytor_Down" := FALSE;
       "Q_Eleveytor_Up" := FALSE;
       "DB_Data".F7.Btt_Down_Selected := FALSE;
   END_IF;
   #_w43 := #_w38 AND "Q_Eleveytor_Up" AND "DB_Data".F7.Btt_Down_Selected AND "M_Check1" AND NOT "DB_Data".F8.Btt_Down_Selected AND NOT "DB_Data".F9.Btt_Down_Selected AND NOT "DB_Data".F10.Btt_Down_Selected AND NOT "DB_Data".F11.Btt_Down_Selected AND NOT "DB_Data".F12.Btt_Down_Selected AND NOT "DB_Data".F13.Btt_Down_Selected AND NOT "DB_Data".F14.Btt_Down_Selected AND NOT "DB_Data".F15.Btt_Down_Selected AND NOT "DB_Data".F16.Btt_Down_Selected AND NOT "DB_Data".F17.Btt_Down_Selected AND NOT "DB_Data".F18.Btt_Down_Selected AND NOT "DB_Data".F19.Btt_Down_Selected AND NOT "DB_Data".F20.Btt_Down_Selected;
   #_w44 := #_w43 AND NOT "P175";   // rising edge
   "P175" := #_w43;
   IF #_w44 THEN
       "Q_Door_Open" := TRUE;
       "Q_Eleveytor_Up" := FALSE;
       "DB_Data".F7.Btt_Down_Selected := FALSE;
   END_IF;
   #_w45 := NOT "AlwaysFALSE" AND "DB_Data".F8.Sensor_Correct_Position;
   #_w46 := #_w45 AND "Q_Eleveytor_Up" AND "DB_Data".F8.Btt_Up_Selected;
   #_w47 := #_w46 AND NOT "P146";   // rising edge
   "P146" := #_w46;
   IF #_w47 THEN
       "Q_Door_Open" := TRUE;
       "Q_Eleveytor_Up" := FALSE;
       "Q_Eleveytor_Down" := FALSE;
       "DB_Data".F8.Btt_Up_Selected := FALSE;
   END_IF;
   #_w48 := #_w45 AND "Q_Eleveytor_Down" AND "DB_Data".F8.Btt_Down_Selected;
   #_w49 := #_w48 AND NOT "P147";   // rising edge
   "P147" := #_w48;
   IF #_w49 THEN
       "Q_Door_Open" := TRUE;
       "Q_Eleveytor_Down" := FALSE;
       "Q_Eleveytor_Up" := FALSE;
       "DB_Data".F8.Btt_Down_Selected := FALSE;
   END_IF;
   #_w50 := #_w45 AND "Q_Eleveytor_Up" AND "DB_Data".F8.Btt_Down_Selected AND "M_Check1" AND NOT "DB_Data".F9.Btt_Down_Selected AND NOT "DB_Data".F10.Btt_Down_Selected AND NOT "DB_Data".F11.Btt_Down_Selected AND NOT "DB_Data".F12.Btt_Down_Selected AND NOT "DB_Data".F13.Btt_Down_Selected AND NOT "DB_Data".F14.Btt_Down_Selected AND NOT "DB_Data".F15.Btt_Down_Selected AND NOT "DB_Data".F16.Btt_Down_Selected AND NOT "DB_Data".F17.Btt_Down_Selected AND NOT "DB_Data".F18.Btt_Down_Selected AND NOT "DB_Data".F19.Btt_Down_Selected AND NOT "DB_Data".F20.Btt_Down_Selected;
   #_w51 := #_w50 AND NOT "P176";   // rising edge
   "P176" := #_w50;
   IF #_w51 THEN
       "Q_Door_Open" := TRUE;
       "Q_Eleveytor_Up" := FALSE;
       "DB_Data".F8.Btt_Down_Selected := FALSE;
   END_IF;
   #_w52 := NOT "AlwaysFALSE" AND "DB_Data".F9.Sensor_Correct_Position;
   #_w53 := #_w52 AND "Q_Eleveytor_Up" AND "DB_Data".F9.Btt_Up_Selected;
   #_w54 := #_w53 AND NOT "P148";   // rising edge
   "P148" := #_w53;
   IF #_w54 THEN
       "Q_Door_Open" := TRUE;
       "Q_Eleveytor_Up" := FALSE;
       "Q_Eleveytor_Down" := FALSE;
       "DB_Data".F9.Btt_Up_Selected := FALSE;
   END_IF;
   #_w55 := #_w52 AND "Q_Eleveytor_Down" AND "DB_Data".F9.Btt_Down_Selected;
   #_w56 := #_w55 AND NOT "P149";   // rising edge
   "P149" := #_w55;
   IF #_w56 THEN
       "Q_Door_Open" := TRUE;
       "Q_Eleveytor_Down" := FALSE;
       "Q_Eleveytor_Up" := FALSE;
       "DB_Data".F9.Btt_Down_Selected := FALSE;
   END_IF;
   #_w57 := #_w52 AND "Q_Eleveytor_Up" AND "DB_Data".F9.Btt_Down_Selected AND "M_Check1" AND NOT "DB_Data".F10.Btt_Down_Selected AND NOT "DB_Data".F11.Btt_Down_Selected AND NOT "DB_Data".F12.Btt_Down_Selected AND NOT "DB_Data".F13.Btt_Down_Selected AND NOT "DB_Data".F14.Btt_Down_Selected AND NOT "DB_Data".F15.Btt_Down_Selected AND NOT "DB_Data".F16.Btt_Down_Selected AND NOT "DB_Data".F17.Btt_Down_Selected AND NOT "DB_Data".F18.Btt_Down_Selected AND NOT "DB_Data".F19.Btt_Down_Selected AND NOT "DB_Data".F20.Btt_Down_Selected;
   #_w58 := #_w57 AND NOT "P177";   // rising edge
   "P177" := #_w57;
   IF #_w58 THEN
       "Q_Door_Open" := TRUE;
       "Q_Eleveytor_Up" := FALSE;
       "DB_Data".F9.Btt_Down_Selected := FALSE;
   END_IF;
   #_w59 := NOT "AlwaysFALSE" AND "DB_Data".F10.Sensor_Correct_Position;
   #_w60 := #_w59 AND "Q_Eleveytor_Up" AND "DB_Data".F10.Btt_Up_Selected;
   #_w61 := #_w60 AND NOT "P150";   // rising edge
   "P150" := #_w60;
   IF #_w61 THEN
       "Q_Door_Open" := TRUE;
       "Q_Eleveytor_Up" := FALSE;
       "Q_Eleveytor_Down" := FALSE;
       "DB_Data".F10.Btt_Up_Selected := FALSE;
   END_IF;
   #_w62 := #_w59 AND "Q_Eleveytor_Down" AND "DB_Data".F10.Btt_Down_Selected;
   #_w63 := #_w62 AND NOT "P48";   // rising edge
   "P48" := #_w62;
   IF #_w63 THEN
       "Q_Door_Open" := TRUE;
       "Q_Eleveytor_Down" := FALSE;
       "Q_Eleveytor_Up" := FALSE;
       "DB_Data".F10.Btt_Down_Selected := FALSE;
   END_IF;
   #_w64 := #_w59 AND "Q_Eleveytor_Up" AND "DB_Data".F10.Btt_Down_Selected AND "M_Check1" AND NOT "DB_Data".F11.Btt_Down_Selected AND NOT "DB_Data".F12.Btt_Down_Selected AND NOT "DB_Data".F13.Btt_Down_Selected AND NOT "DB_Data".F14.Btt_Down_Selected AND NOT "DB_Data".F15.Btt_Down_Selected AND NOT "DB_Data".F16.Btt_Down_Selected AND NOT "DB_Data".F17.Btt_Down_Selected AND NOT "DB_Data".F18.Btt_Down_Selected AND NOT "DB_Data".F19.Btt_Down_Selected AND NOT "DB_Data".F20.Btt_Down_Selected;
   #_w65 := #_w64 AND NOT "P178";   // rising edge
   "P178" := #_w64;
   IF #_w65 THEN
       "Q_Door_Open" := TRUE;
       "Q_Eleveytor_Up" := FALSE;
       "DB_Data".F10.Btt_Down_Selected := FALSE;
   END_IF;
   #_w66 := NOT "AlwaysFALSE" AND "DB_Data".F11.Sensor_Correct_Position;
   #_w67 := #_w66 AND "Q_Eleveytor_Up" AND "DB_Data".F11.Btt_Up_Selected;
   #_w68 := #_w67 AND NOT "P151";   // rising edge
   "P151" := #_w67;
   IF #_w68 THEN
       "Q_Door_Open" := TRUE;
       "Q_Eleveytor_Up" := FALSE;
       "Q_Eleveytor_Down" := FALSE;
       "DB_Data".F11.Btt_Up_Selected := FALSE;
   END_IF;
   #_w69 := #_w66 AND "Q_Eleveytor_Down" AND "DB_Data".F11.Btt_Down_Selected;
   #_w70 := #_w69 AND NOT "P152";   // rising edge
   "P152" := #_w69;
   IF #_w70 THEN
       "Q_Door_Open" := TRUE;
       "Q_Eleveytor_Down" := FALSE;
       "Q_Eleveytor_Up" := FALSE;
       "DB_Data".F11.Btt_Down_Selected := FALSE;
   END_IF;
   #_w71 := #_w66 AND "Q_Eleveytor_Up" AND "DB_Data".F11.Btt_Down_Selected AND "M_Check1" AND NOT "DB_Data".F12.Btt_Down_Selected AND NOT "DB_Data".F13.Btt_Down_Selected AND NOT "DB_Data".F14.Btt_Down_Selected AND NOT "DB_Data".F15.Btt_Down_Selected AND NOT "DB_Data".F16.Btt_Down_Selected AND NOT "DB_Data".F17.Btt_Down_Selected AND NOT "DB_Data".F18.Btt_Down_Selected AND NOT "DB_Data".F19.Btt_Down_Selected AND NOT "DB_Data".F20.Btt_Down_Selected;
   #_w72 := #_w71 AND NOT "P179";   // rising edge
   "P179" := #_w71;
   IF #_w72 THEN
       "Q_Door_Open" := TRUE;
       "Q_Eleveytor_Up" := FALSE;
       "DB_Data".F11.Btt_Down_Selected := FALSE;
   END_IF;
   #_w73 := NOT "AlwaysFALSE" AND "DB_Data".F12.Sensor_Correct_Position;
   #_w74 := #_w73 AND "Q_Eleveytor_Up" AND "DB_Data".F12.Btt_Up_Selected;
   #_w75 := #_w74 AND NOT "P153";   // rising edge
   "P153" := #_w74;
   IF #_w75 THEN
       "Q_Door_Open" := TRUE;
       "Q_Eleveytor_Up" := FALSE;
       "Q_Eleveytor_Down" := FALSE;
       "DB_Data".F12.Btt_Up_Selected := FALSE;
   END_IF;
   #_w76 := #_w73 AND "Q_Eleveytor_Down" AND "DB_Data".F12.Btt_Down_Selected;
   #_w77 := #_w76 AND NOT "P154";   // rising edge
   "P154" := #_w76;
   IF #_w77 THEN
       "Q_Door_Open" := TRUE;
       "Q_Eleveytor_Down" := FALSE;
       "Q_Eleveytor_Up" := FALSE;
       "DB_Data".F12.Btt_Down_Selected := FALSE;
   END_IF;
   #_w78 := #_w73 AND "Q_Eleveytor_Up" AND "DB_Data".F12.Btt_Down_Selected AND "M_Check1" AND NOT "DB_Data".F13.Btt_Down_Selected AND NOT "DB_Data".F14.Btt_Down_Selected AND NOT "DB_Data".F15.Btt_Down_Selected AND NOT "DB_Data".F16.Btt_Down_Selected AND NOT "DB_Data".F17.Btt_Down_Selected AND NOT "DB_Data".F18.Btt_Down_Selected AND NOT "DB_Data".F19.Btt_Down_Selected AND NOT "DB_Data".F20.Btt_Down_Selected;
   #_w79 := #_w78 AND NOT "P180";   // rising edge
   "P180" := #_w78;
   IF #_w79 THEN
       "Q_Door_Open" := TRUE;
       "Q_Eleveytor_Up" := FALSE;
       "DB_Data".F12.Btt_Down_Selected := FALSE;
   END_IF;
   #_w80 := NOT "AlwaysFALSE" AND "DB_Data".F13.Sensor_Correct_Position;
   #_w81 := #_w80 AND "Q_Eleveytor_Up" AND "DB_Data".F13.Btt_Up_Selected;
   #_w82 := #_w81 AND NOT "P155";   // rising edge
   "P155" := #_w81;
   IF #_w82 THEN
       "Q_Door_Open" := TRUE;
       "Q_Eleveytor_Up" := FALSE;
       "Q_Eleveytor_Down" := FALSE;
       "DB_Data".F13.Btt_Up_Selected := FALSE;
   END_IF;
   #_w83 := #_w80 AND "Q_Eleveytor_Down" AND "DB_Data".F13.Btt_Down_Selected;
   #_w84 := #_w83 AND NOT "P156";   // rising edge
   "P156" := #_w83;
   IF #_w84 THEN
       "Q_Door_Open" := TRUE;
       "Q_Eleveytor_Down" := FALSE;
       "Q_Eleveytor_Up" := FALSE;
       "DB_Data".F13.Btt_Down_Selected := FALSE;
   END_IF;
   #_w85 := #_w80 AND "Q_Eleveytor_Up" AND "DB_Data".F13.Btt_Down_Selected AND "M_Check1" AND NOT "DB_Data".F14.Btt_Down_Selected AND NOT "DB_Data".F15.Btt_Down_Selected AND NOT "DB_Data".F16.Btt_Down_Selected AND NOT "DB_Data".F17.Btt_Down_Selected AND NOT "DB_Data".F18.Btt_Down_Selected AND NOT "DB_Data".F19.Btt_Down_Selected AND NOT "DB_Data".F20.Btt_Down_Selected;
   #_w86 := #_w85 AND NOT "P181";   // rising edge
   "P181" := #_w85;
   IF #_w86 THEN
       "Q_Door_Open" := TRUE;
       "Q_Eleveytor_Up" := FALSE;
       "DB_Data".F13.Btt_Down_Selected := FALSE;
   END_IF;
   #_w87 := NOT "AlwaysFALSE" AND "DB_Data".F14.Sensor_Correct_Position;
   #_w88 := #_w87 AND "Q_Eleveytor_Up" AND "DB_Data".F14.Btt_Up_Selected;
   #_w89 := #_w88 AND NOT "P157";   // rising edge
   "P157" := #_w88;
   IF #_w89 THEN
       "Q_Door_Open" := TRUE;
       "Q_Eleveytor_Up" := FALSE;
       "Q_Eleveytor_Down" := FALSE;
       "DB_Data".F14.Btt_Up_Selected := FALSE;
   END_IF;
   #_w90 := #_w87 AND "Q_Eleveytor_Down" AND "DB_Data".F14.Btt_Down_Selected;
   #_w91 := #_w90 AND NOT "P158";   // rising edge
   "P158" := #_w90;
   IF #_w91 THEN
       "Q_Door_Open" := TRUE;
       "Q_Eleveytor_Down" := FALSE;
       "Q_Eleveytor_Up" := FALSE;
       "DB_Data".F14.Btt_Down_Selected := FALSE;
   END_IF;
   #_w92 := #_w87 AND "Q_Eleveytor_Up" AND "DB_Data".F14.Btt_Down_Selected AND "M_Check1" AND NOT "DB_Data".F15.Btt_Down_Selected AND NOT "DB_Data".F16.Btt_Down_Selected AND NOT "DB_Data".F17.Btt_Down_Selected AND NOT "DB_Data".F18.Btt_Down_Selected AND NOT "DB_Data".F19.Btt_Down_Selected AND NOT "DB_Data".F20.Btt_Down_Selected;
   #_w93 := #_w92 AND NOT "P182";   // rising edge
   "P182" := #_w92;
   IF #_w93 THEN
       "Q_Door_Open" := TRUE;
       "Q_Eleveytor_Up" := FALSE;
       "DB_Data".F14.Btt_Down_Selected := FALSE;
   END_IF;
   #_w94 := NOT "AlwaysFALSE" AND "DB_Data".F15.Sensor_Correct_Position;
   #_w95 := #_w94 AND "Q_Eleveytor_Up" AND "DB_Data".F15.Btt_Up_Selected;
   #_w96 := #_w95 AND NOT "P159";   // rising edge
   "P159" := #_w95;
   IF #_w96 THEN
       "Q_Door_Open" := TRUE;
       "Q_Eleveytor_Up" := FALSE;
       "Q_Eleveytor_Down" := FALSE;
       "DB_Data".F15.Btt_Up_Selected := FALSE;
   END_IF;
   #_w97 := #_w94 AND "Q_Eleveytor_Down" AND "DB_Data".F15.Btt_Down_Selected;
   #_w98 := #_w97 AND NOT "P160";   // rising edge
   "P160" := #_w97;
   IF #_w98 THEN
       "Q_Door_Open" := TRUE;
       "Q_Eleveytor_Down" := FALSE;
       "Q_Eleveytor_Up" := FALSE;
       "DB_Data".F15.Btt_Down_Selected := FALSE;
   END_IF;
   #_w99 := #_w94 AND "Q_Eleveytor_Up" AND "DB_Data".F15.Btt_Down_Selected AND "M_Check1" AND NOT "DB_Data".F16.Btt_Down_Selected AND NOT "DB_Data".F17.Btt_Down_Selected AND NOT "DB_Data".F18.Btt_Down_Selected AND NOT "DB_Data".F19.Btt_Down_Selected AND NOT "DB_Data".F20.Btt_Down_Selected;
   #_w100 := #_w99 AND NOT "P183";   // rising edge
   "P183" := #_w99;
   IF #_w100 THEN
       "Q_Door_Open" := TRUE;
       "Q_Eleveytor_Up" := FALSE;
       "DB_Data".F15.Btt_Down_Selected := FALSE;
   END_IF;
   #_w101 := NOT "AlwaysFALSE" AND "DB_Data".F16.Sensor_Correct_Position;
   #_w102 := #_w101 AND "Q_Eleveytor_Up" AND "DB_Data".F16.Btt_Up_Selected;
   #_w103 := #_w102 AND NOT "P161";   // rising edge
   "P161" := #_w102;
   IF #_w103 THEN
       "Q_Door_Open" := TRUE;
       "Q_Eleveytor_Up" := FALSE;
       "Q_Eleveytor_Down" := FALSE;
       "DB_Data".F16.Btt_Up_Selected := FALSE;
   END_IF;
   #_w104 := #_w101 AND "Q_Eleveytor_Down" AND "DB_Data".F16.Btt_Down_Selected;
   #_w105 := #_w104 AND NOT "P162";   // rising edge
   "P162" := #_w104;
   IF #_w105 THEN
       "Q_Door_Open" := TRUE;
       "Q_Eleveytor_Down" := FALSE;
       "Q_Eleveytor_Up" := FALSE;
       "DB_Data".F16.Btt_Down_Selected := FALSE;
   END_IF;
   #_w106 := #_w101 AND "Q_Eleveytor_Up" AND "DB_Data".F16.Btt_Down_Selected AND "M_Check1" AND NOT "DB_Data".F17.Btt_Down_Selected AND NOT "DB_Data".F18.Btt_Down_Selected AND NOT "DB_Data".F19.Btt_Down_Selected AND NOT "DB_Data".F20.Btt_Down_Selected;
   #_w107 := #_w106 AND NOT "P183";   // rising edge
   "P183" := #_w106;
   IF #_w107 THEN
       "Q_Door_Open" := TRUE;
       "Q_Eleveytor_Up" := FALSE;
       "DB_Data".F16.Btt_Down_Selected := FALSE;
   END_IF;
   #_w108 := NOT "AlwaysFALSE" AND "DB_Data".F17.Sensor_Correct_Position;
   #_w109 := #_w108 AND "Q_Eleveytor_Up" AND "DB_Data".F17.Btt_Up_Selected;
   #_w110 := #_w109 AND NOT "P163";   // rising edge
   "P163" := #_w109;
   IF #_w110 THEN
       "Q_Door_Open" := TRUE;
       "Q_Eleveytor_Up" := FALSE;
       "Q_Eleveytor_Down" := FALSE;
       "DB_Data".F17.Btt_Up_Selected := FALSE;
   END_IF;
   #_w111 := #_w108 AND "Q_Eleveytor_Down" AND "DB_Data".F17.Btt_Down_Selected;
   #_w112 := #_w111 AND NOT "P164";   // rising edge
   "P164" := #_w111;
   IF #_w112 THEN
       "Q_Door_Open" := TRUE;
       "Q_Eleveytor_Down" := FALSE;
       "Q_Eleveytor_Up" := FALSE;
       "DB_Data".F17.Btt_Down_Selected := FALSE;
   END_IF;
   #_w113 := #_w108 AND "Q_Eleveytor_Up" AND "DB_Data".F17.Btt_Down_Selected AND "M_Check1" AND NOT "DB_Data".F18.Btt_Down_Selected AND NOT "DB_Data".F19.Btt_Down_Selected AND NOT "DB_Data".F20.Btt_Down_Selected;
   #_w114 := #_w113 AND NOT "P184";   // rising edge
   "P184" := #_w113;
   IF #_w114 THEN
       "Q_Door_Open" := TRUE;
       "Q_Eleveytor_Up" := FALSE;
       "DB_Data".F17.Btt_Down_Selected := FALSE;
   END_IF;
   #_w115 := NOT "AlwaysFALSE" AND "DB_Data".F18.Sensor_Correct_Position;
   #_w116 := #_w115 AND "Q_Eleveytor_Up" AND "DB_Data".F18.Btt_Up_Selected;
   #_w117 := #_w116 AND NOT "P165";   // rising edge
   "P165" := #_w116;
   IF #_w117 THEN
       "Q_Door_Open" := TRUE;
       "Q_Eleveytor_Up" := FALSE;
       "Q_Eleveytor_Down" := FALSE;
       "DB_Data".F18.Btt_Up_Selected := FALSE;
   END_IF;
   #_w118 := #_w115 AND "Q_Eleveytor_Down" AND "DB_Data".F18.Btt_Down_Selected;
   #_w119 := #_w118 AND NOT "P166";   // rising edge
   "P166" := #_w118;
   IF #_w119 THEN
       "Q_Door_Open" := TRUE;
       "Q_Eleveytor_Down" := FALSE;
       "Q_Eleveytor_Up" := FALSE;
       "DB_Data".F18.Btt_Down_Selected := FALSE;
   END_IF;
   #_w120 := #_w115 AND "Q_Eleveytor_Up" AND "DB_Data".F18.Btt_Down_Selected AND "M_Check1" AND NOT "DB_Data".F19.Btt_Down_Selected AND NOT "DB_Data".F20.Btt_Down_Selected;
   #_w121 := #_w120 AND NOT "P185";   // rising edge
   "P185" := #_w120;
   IF #_w121 THEN
       "Q_Door_Open" := TRUE;
       "Q_Eleveytor_Up" := FALSE;
       "DB_Data".F18.Btt_Down_Selected := FALSE;
   END_IF;
   #_w122 := NOT "AlwaysFALSE" AND "DB_Data".F19.Sensor_Correct_Position;
   #_w123 := #_w122 AND "Q_Eleveytor_Up" AND "DB_Data".F19.Btt_Up_Selected;
   #_w124 := #_w123 AND NOT "P167";   // rising edge
   "P167" := #_w123;
   IF #_w124 THEN
       "Q_Door_Open" := TRUE;
       "Q_Eleveytor_Up" := FALSE;
       "Q_Eleveytor_Down" := FALSE;
       "DB_Data".F19.Btt_Up_Selected := FALSE;
   END_IF;
   #_w125 := #_w122 AND "Q_Eleveytor_Down" AND "DB_Data".F19.Btt_Down_Selected;
   #_w126 := #_w125 AND NOT "P168";   // rising edge
   "P168" := #_w125;
   IF #_w126 THEN
       "Q_Door_Open" := TRUE;
       "Q_Eleveytor_Down" := FALSE;
       "Q_Eleveytor_Up" := FALSE;
       "DB_Data".F19.Btt_Down_Selected := FALSE;
   END_IF;
   #_w127 := #_w122 AND "Q_Eleveytor_Up" AND "DB_Data".F19.Btt_Down_Selected AND "M_Check1" AND NOT "DB_Data".F20.Btt_Down_Selected;
   #_w128 := #_w127 AND NOT "P186";   // rising edge
   "P186" := #_w127;
   IF #_w128 THEN
       "Q_Door_Open" := TRUE;
       "Q_Eleveytor_Up" := FALSE;
       "DB_Data".F19.Btt_Down_Selected := FALSE;
   END_IF;
   #_w129 := NOT "AlwaysFALSE" AND "DB_Data".F20.Sensor_Correct_Position AND "Q_Eleveytor_Up" AND "DB_Data".F20.Btt_Down_Selected;
   #_w130 := #_w129 AND NOT "P169";   // rising edge
   "P169" := #_w129;
   IF #_w130 THEN
       "Q_Door_Open" := TRUE;
       "Q_Eleveytor_Up" := FALSE;
       "DB_Data".F20.Btt_Down_Selected := FALSE;
   END_IF;
END_REGION

REGION Network 25: Tự động đóng cửa
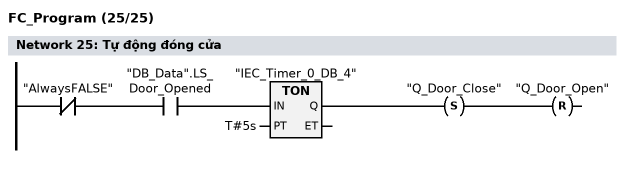
   "IEC_Timer_0_DB_4".TON(IN := NOT "AlwaysFALSE" AND "DB_Data".LS_Door_Opened, PT := T#5s);
   IF "IEC_Timer_0_DB_4".Q THEN
       "Q_Door_Close" := TRUE;
       "Q_Door_Open" := FALSE;
   END_IF;
END_REGION
END_FUNCTION

FUNCTION "FC_Simulation" : Void   // FC3, LAD
{ S7_Optimized_Access := 'TRUE' }
VERSION : 0.1
   VAR_TEMP   // added for the SCL form of the ladder/FBD networks
      _w1 : Bool;
      _w2 : Bool;
      _w3 : Bool;
      _w4 : Bool;
      _w5 : Bool;
   END_VAR
BEGIN

REGION Network 1: Thang chuyển động lên xuống
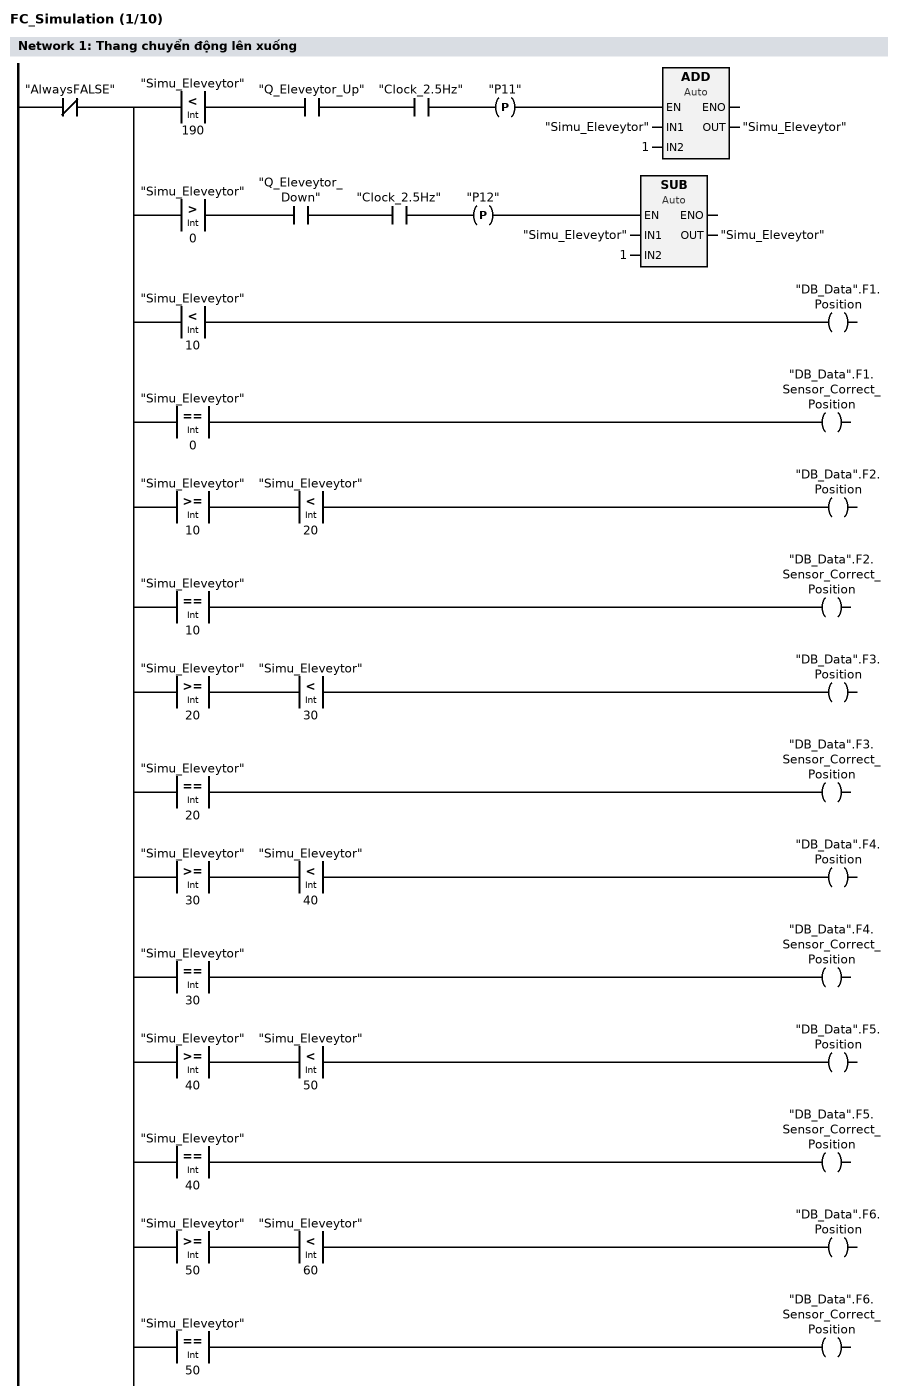
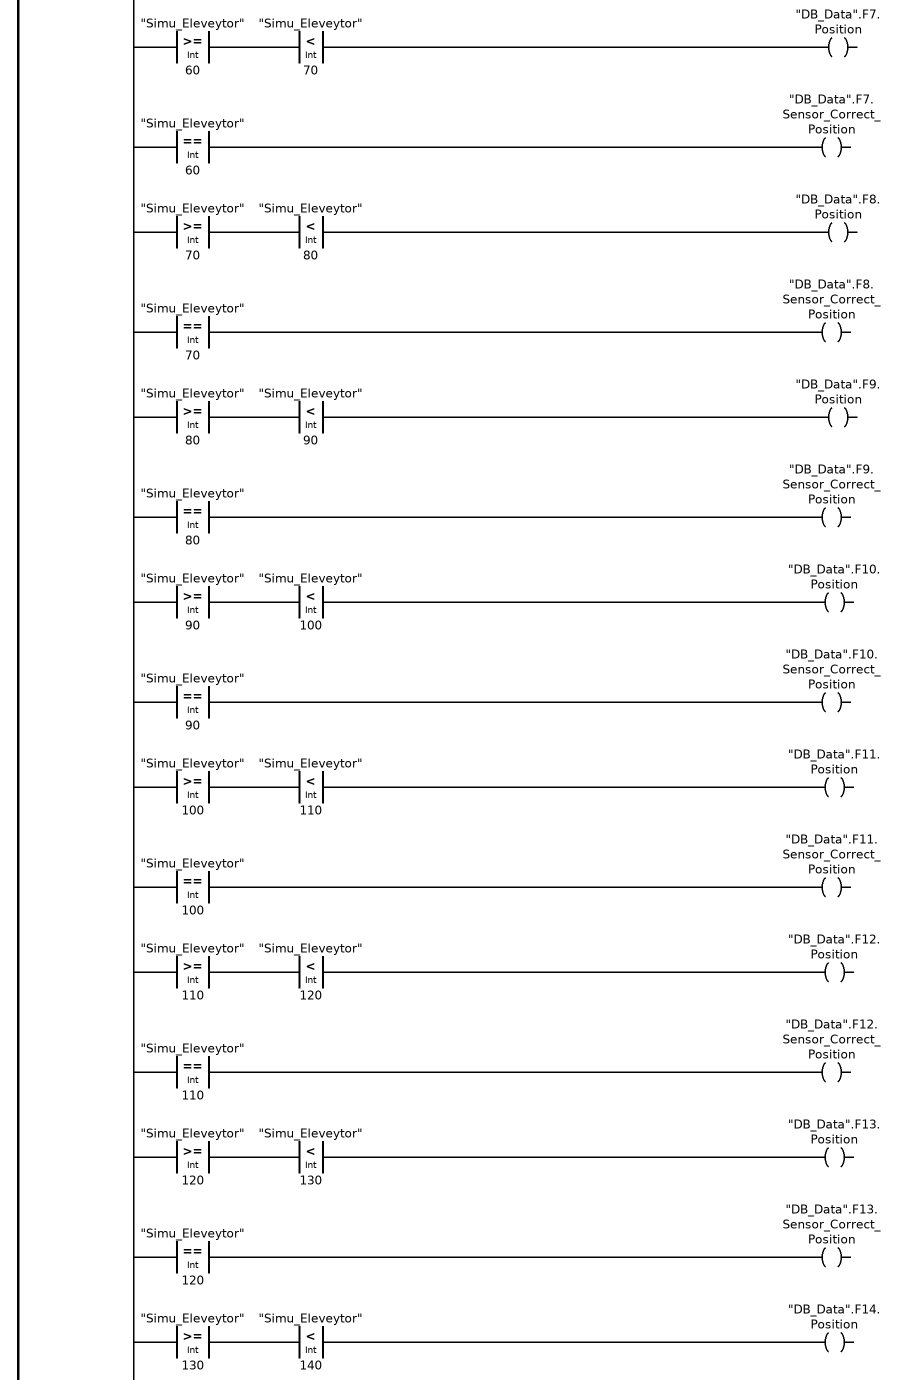
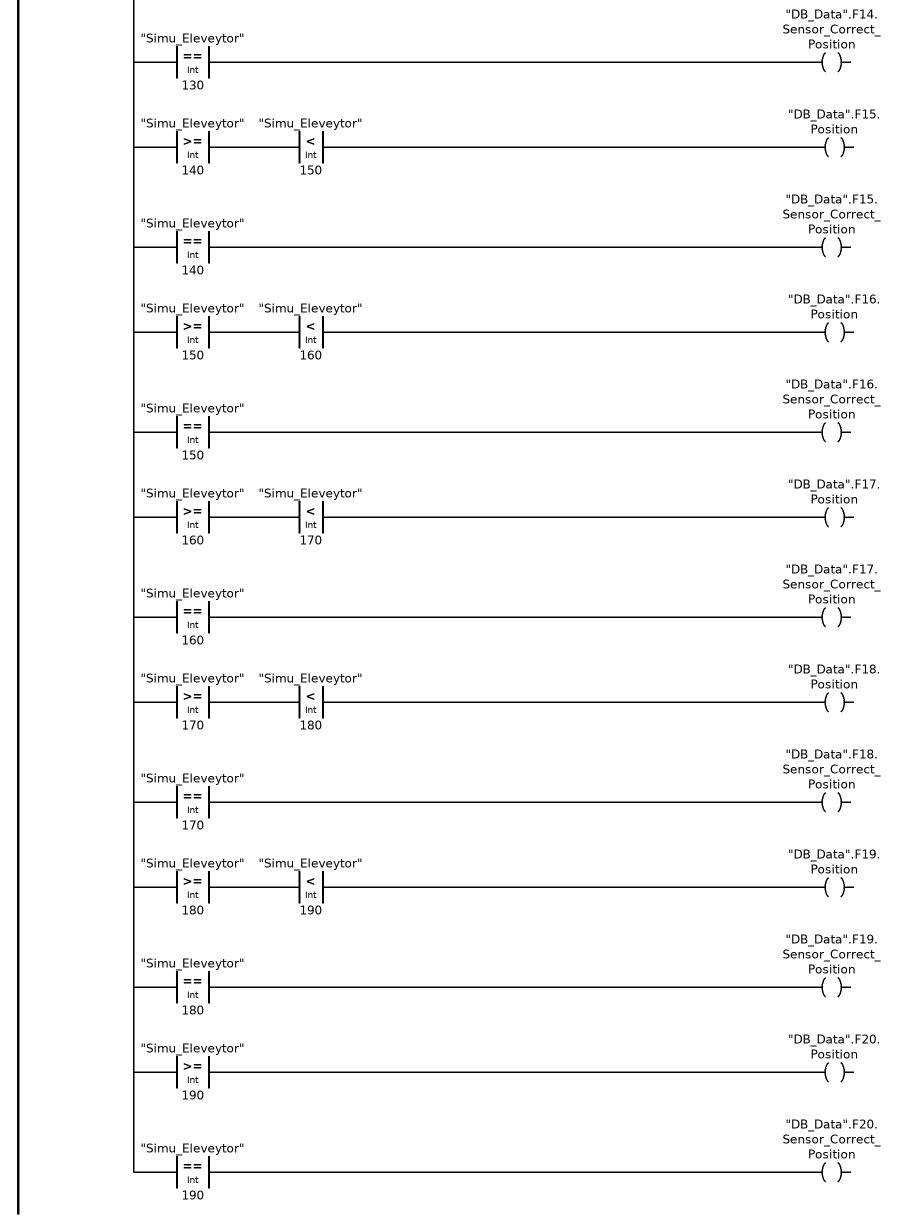
   RUNG wire#powerrail
      I_Contact( "AlwaysFALSE" )
      wire#w1
      { S7_Templates := "SrcType := Int" } LT_Contact(in1 := "Simu_Eleveytor", in2 := 190)
      Contact( "Q_Eleveytor_Up" )
      Contact( "Clock_2.5Hz" )
      P_Trig( "P11" )
      Add(in1 := "Simu_Eleveytor", in2 := 1, out => "Simu_Eleveytor")
   END_RUNG
   RUNG wire#w1
      { S7_Templates := "SrcType := Int" } GT_Contact(in1 := "Simu_Eleveytor", in2 := 0)
      Contact( "Q_Eleveytor_Down" )
      Contact( "Clock_2.5Hz" )
      P_Trig( "P12" )
      Sub(in1 := "Simu_Eleveytor", in2 := 1, out => "Simu_Eleveytor")
   END_RUNG
   RUNG wire#w1
      { S7_Templates := "SrcType := Int" } LT_Contact(in1 := "Simu_Eleveytor", in2 := 10)
      Coil( "DB_Data".F1.Position )
   END_RUNG
   RUNG wire#w1
      { S7_Templates := "SrcType := Int" } EQ_Contact(in1 := "Simu_Eleveytor", in2 := 0)
      Coil( "DB_Data".F1.Sensor_Correct_Position )
   END_RUNG
   RUNG wire#w1
      { S7_Templates := "SrcType := Int" } GE_Contact(in1 := "Simu_Eleveytor", in2 := 10)
      { S7_Templates := "SrcType := Int" } LT_Contact(in1 := "Simu_Eleveytor", in2 := 20)
      Coil( "DB_Data".F2.Position )
   END_RUNG
   RUNG wire#w1
      { S7_Templates := "SrcType := Int" } EQ_Contact(in1 := "Simu_Eleveytor", in2 := 10)
      Coil( "DB_Data".F2.Sensor_Correct_Position )
   END_RUNG
   RUNG wire#w1
      { S7_Templates := "SrcType := Int" } GE_Contact(in1 := "Simu_Eleveytor", in2 := 20)
      { S7_Templates := "SrcType := Int" } LT_Contact(in1 := "Simu_Eleveytor", in2 := 30)
      Coil( "DB_Data".F3.Position )
   END_RUNG
   RUNG wire#w1
      { S7_Templates := "SrcType := Int" } EQ_Contact(in1 := "Simu_Eleveytor", in2 := 20)
      Coil( "DB_Data".F3.Sensor_Correct_Position )
   END_RUNG
   RUNG wire#w1
      { S7_Templates := "SrcType := Int" } GE_Contact(in1 := "Simu_Eleveytor", in2 := 30)
      { S7_Templates := "SrcType := Int" } LT_Contact(in1 := "Simu_Eleveytor", in2 := 40)
      Coil( "DB_Data".F4.Position )
   END_RUNG
   RUNG wire#w1
      { S7_Templates := "SrcType := Int" } EQ_Contact(in1 := "Simu_Eleveytor", in2 := 30)
      Coil( "DB_Data".F4.Sensor_Correct_Position )
   END_RUNG
   RUNG wire#w1
      { S7_Templates := "SrcType := Int" } GE_Contact(in1 := "Simu_Eleveytor", in2 := 40)
      { S7_Templates := "SrcType := Int" } LT_Contact(in1 := "Simu_Eleveytor", in2 := 50)
      Coil( "DB_Data".F5.Position )
   END_RUNG
   RUNG wire#w1
      { S7_Templates := "SrcType := Int" } EQ_Contact(in1 := "Simu_Eleveytor", in2 := 40)
      Coil( "DB_Data".F5.Sensor_Correct_Position )
   END_RUNG
   RUNG wire#w1
      { S7_Templates := "SrcType := Int" } GE_Contact(in1 := "Simu_Eleveytor", in2 := 50)
      { S7_Templates := "SrcType := Int" } LT_Contact(in1 := "Simu_Eleveytor", in2 := 60)
      Coil( "DB_Data".F6.Position )
   END_RUNG
   RUNG wire#w1
      { S7_Templates := "SrcType := Int" } EQ_Contact(in1 := "Simu_Eleveytor", in2 := 50)
      Coil( "DB_Data".F6.Sensor_Correct_Position )
   END_RUNG
   RUNG wire#w1
      { S7_Templates := "SrcType := Int" } GE_Contact(in1 := "Simu_Eleveytor", in2 := 60)
      { S7_Templates := "SrcType := Int" } LT_Contact(in1 := "Simu_Eleveytor", in2 := 70)
      Coil( "DB_Data".F7.Position )
   END_RUNG
   RUNG wire#w1
      { S7_Templates := "SrcType := Int" } EQ_Contact(in1 := "Simu_Eleveytor", in2 := 60)
      Coil( "DB_Data".F7.Sensor_Correct_Position )
   END_RUNG
   RUNG wire#w1
      { S7_Templates := "SrcType := Int" } GE_Contact(in1 := "Simu_Eleveytor", in2 := 70)
      { S7_Templates := "SrcType := Int" } LT_Contact(in1 := "Simu_Eleveytor", in2 := 80)
      Coil( "DB_Data".F8.Position )
   END_RUNG
   RUNG wire#w1
      { S7_Templates := "SrcType := Int" } EQ_Contact(in1 := "Simu_Eleveytor", in2 := 70)
      Coil( "DB_Data".F8.Sensor_Correct_Position )
   END_RUNG
   RUNG wire#w1
      { S7_Templates := "SrcType := Int" } GE_Contact(in1 := "Simu_Eleveytor", in2 := 80)
      { S7_Templates := "SrcType := Int" } LT_Contact(in1 := "Simu_Eleveytor", in2 := 90)
      Coil( "DB_Data".F9.Position )
   END_RUNG
   RUNG wire#w1
      { S7_Templates := "SrcType := Int" } EQ_Contact(in1 := "Simu_Eleveytor", in2 := 80)
      Coil( "DB_Data".F9.Sensor_Correct_Position )
   END_RUNG
   RUNG wire#w1
      { S7_Templates := "SrcType := Int" } GE_Contact(in1 := "Simu_Eleveytor", in2 := 90)
      { S7_Templates := "SrcType := Int" } LT_Contact(in1 := "Simu_Eleveytor", in2 := 100)
      Coil( "DB_Data".F10.Position )
   END_RUNG
   RUNG wire#w1
      { S7_Templates := "SrcType := Int" } EQ_Contact(in1 := "Simu_Eleveytor", in2 := 90)
      Coil( "DB_Data".F10.Sensor_Correct_Position )
   END_RUNG
   RUNG wire#w1
      { S7_Templates := "SrcType := Int" } GE_Contact(in1 := "Simu_Eleveytor", in2 := 100)
      { S7_Templates := "SrcType := Int" } LT_Contact(in1 := "Simu_Eleveytor", in2 := 110)
      Coil( "DB_Data".F11.Position )
   END_RUNG
   RUNG wire#w1
      { S7_Templates := "SrcType := Int" } EQ_Contact(in1 := "Simu_Eleveytor", in2 := 100)
      Coil( "DB_Data".F11.Sensor_Correct_Position )
   END_RUNG
   RUNG wire#w1
      { S7_Templates := "SrcType := Int" } GE_Contact(in1 := "Simu_Eleveytor", in2 := 110)
      { S7_Templates := "SrcType := Int" } LT_Contact(in1 := "Simu_Eleveytor", in2 := 120)
      Coil( "DB_Data".F12.Position )
   END_RUNG
   RUNG wire#w1
      { S7_Templates := "SrcType := Int" } EQ_Contact(in1 := "Simu_Eleveytor", in2 := 110)
      Coil( "DB_Data".F12.Sensor_Correct_Position )
   END_RUNG
   RUNG wire#w1
      { S7_Templates := "SrcType := Int" } GE_Contact(in1 := "Simu_Eleveytor", in2 := 120)
      { S7_Templates := "SrcType := Int" } LT_Contact(in1 := "Simu_Eleveytor", in2 := 130)
      Coil( "DB_Data".F13.Position )
   END_RUNG
   RUNG wire#w1
      { S7_Templates := "SrcType := Int" } EQ_Contact(in1 := "Simu_Eleveytor", in2 := 120)
      Coil( "DB_Data".F13.Sensor_Correct_Position )
   END_RUNG
   RUNG wire#w1
      { S7_Templates := "SrcType := Int" } GE_Contact(in1 := "Simu_Eleveytor", in2 := 130)
      { S7_Templates := "SrcType := Int" } LT_Contact(in1 := "Simu_Eleveytor", in2 := 140)
      Coil( "DB_Data".F14.Position )
   END_RUNG
   RUNG wire#w1
      { S7_Templates := "SrcType := Int" } EQ_Contact(in1 := "Simu_Eleveytor", in2 := 130)
      Coil( "DB_Data".F14.Sensor_Correct_Position )
   END_RUNG
   RUNG wire#w1
      { S7_Templates := "SrcType := Int" } GE_Contact(in1 := "Simu_Eleveytor", in2 := 140)
      { S7_Templates := "SrcType := Int" } LT_Contact(in1 := "Simu_Eleveytor", in2 := 150)
      Coil( "DB_Data".F15.Position )
   END_RUNG
   RUNG wire#w1
      { S7_Templates := "SrcType := Int" } EQ_Contact(in1 := "Simu_Eleveytor", in2 := 140)
      Coil( "DB_Data".F15.Sensor_Correct_Position )
   END_RUNG
   RUNG wire#w1
      { S7_Templates := "SrcType := Int" } GE_Contact(in1 := "Simu_Eleveytor", in2 := 150)
      { S7_Templates := "SrcType := Int" } LT_Contact(in1 := "Simu_Eleveytor", in2 := 160)
      Coil( "DB_Data".F16.Position )
   END_RUNG
   RUNG wire#w1
      { S7_Templates := "SrcType := Int" } EQ_Contact(in1 := "Simu_Eleveytor", in2 := 150)
      Coil( "DB_Data".F16.Sensor_Correct_Position )
   END_RUNG
   RUNG wire#w1
      { S7_Templates := "SrcType := Int" } GE_Contact(in1 := "Simu_Eleveytor", in2 := 160)
      { S7_Templates := "SrcType := Int" } LT_Contact(in1 := "Simu_Eleveytor", in2 := 170)
      Coil( "DB_Data".F17.Position )
   END_RUNG
   RUNG wire#w1
      { S7_Templates := "SrcType := Int" } EQ_Contact(in1 := "Simu_Eleveytor", in2 := 160)
      Coil( "DB_Data".F17.Sensor_Correct_Position )
   END_RUNG
   RUNG wire#w1
      { S7_Templates := "SrcType := Int" } GE_Contact(in1 := "Simu_Eleveytor", in2 := 170)
      { S7_Templates := "SrcType := Int" } LT_Contact(in1 := "Simu_Eleveytor", in2 := 180)
      Coil( "DB_Data".F18.Position )
   END_RUNG
   RUNG wire#w1
      { S7_Templates := "SrcType := Int" } EQ_Contact(in1 := "Simu_Eleveytor", in2 := 170)
      Coil( "DB_Data".F18.Sensor_Correct_Position )
   END_RUNG
   RUNG wire#w1
      { S7_Templates := "SrcType := Int" } GE_Contact(in1 := "Simu_Eleveytor", in2 := 180)
      { S7_Templates := "SrcType := Int" } LT_Contact(in1 := "Simu_Eleveytor", in2 := 190)
      Coil( "DB_Data".F19.Position )
   END_RUNG
   RUNG wire#w1
      { S7_Templates := "SrcType := Int" } EQ_Contact(in1 := "Simu_Eleveytor", in2 := 180)
      Coil( "DB_Data".F19.Sensor_Correct_Position )
   END_RUNG
   RUNG wire#w1
      { S7_Templates := "SrcType := Int" } GE_Contact(in1 := "Simu_Eleveytor", in2 := 190)
      Coil( "DB_Data".F20.Position )
   END_RUNG
   RUNG wire#w1
      { S7_Templates := "SrcType := Int" } EQ_Contact(in1 := "Simu_Eleveytor", in2 := 190)
      Coil( "DB_Data".F20.Sensor_Correct_Position )
   END_RUNG
   // the same network as SCL:
   #_w1 := NOT "AlwaysFALSE" AND ("Simu_Eleveytor" < 190) AND "Q_Eleveytor_Up" AND "Clock_2.5Hz";
   #_w2 := #_w1 AND NOT "P11";   // rising edge
   "P11" := #_w1;
   IF #_w2 THEN "Simu_Eleveytor" := "Simu_Eleveytor" + 1; END_IF;
   #_w3 := NOT "AlwaysFALSE" AND ("Simu_Eleveytor" > 0) AND "Q_Eleveytor_Down" AND "Clock_2.5Hz";
   #_w4 := #_w3 AND NOT "P12";   // rising edge
   "P12" := #_w3;
   IF #_w4 THEN "Simu_Eleveytor" := "Simu_Eleveytor" - 1; END_IF;
   "DB_Data".F1.Position := NOT "AlwaysFALSE" AND ("Simu_Eleveytor" < 10);
   "DB_Data".F1.Sensor_Correct_Position := NOT "AlwaysFALSE" AND ("Simu_Eleveytor" = 0);
   "DB_Data".F2.Position := NOT "AlwaysFALSE" AND ("Simu_Eleveytor" >= 10) AND ("Simu_Eleveytor" < 20);
   "DB_Data".F2.Sensor_Correct_Position := NOT "AlwaysFALSE" AND ("Simu_Eleveytor" = 10);
   "DB_Data".F3.Position := NOT "AlwaysFALSE" AND ("Simu_Eleveytor" >= 20) AND ("Simu_Eleveytor" < 30);
   "DB_Data".F3.Sensor_Correct_Position := NOT "AlwaysFALSE" AND ("Simu_Eleveytor" = 20);
   "DB_Data".F4.Position := NOT "AlwaysFALSE" AND ("Simu_Eleveytor" >= 30) AND ("Simu_Eleveytor" < 40);
   "DB_Data".F4.Sensor_Correct_Position := NOT "AlwaysFALSE" AND ("Simu_Eleveytor" = 30);
   "DB_Data".F5.Position := NOT "AlwaysFALSE" AND ("Simu_Eleveytor" >= 40) AND ("Simu_Eleveytor" < 50);
   "DB_Data".F5.Sensor_Correct_Position := NOT "AlwaysFALSE" AND ("Simu_Eleveytor" = 40);
   "DB_Data".F6.Position := NOT "AlwaysFALSE" AND ("Simu_Eleveytor" >= 50) AND ("Simu_Eleveytor" < 60);
   "DB_Data".F6.Sensor_Correct_Position := NOT "AlwaysFALSE" AND ("Simu_Eleveytor" = 50);
   "DB_Data".F7.Position := NOT "AlwaysFALSE" AND ("Simu_Eleveytor" >= 60) AND ("Simu_Eleveytor" < 70);
   "DB_Data".F7.Sensor_Correct_Position := NOT "AlwaysFALSE" AND ("Simu_Eleveytor" = 60);
   "DB_Data".F8.Position := NOT "AlwaysFALSE" AND ("Simu_Eleveytor" >= 70) AND ("Simu_Eleveytor" < 80);
   "DB_Data".F8.Sensor_Correct_Position := NOT "AlwaysFALSE" AND ("Simu_Eleveytor" = 70);
   "DB_Data".F9.Position := NOT "AlwaysFALSE" AND ("Simu_Eleveytor" >= 80) AND ("Simu_Eleveytor" < 90);
   "DB_Data".F9.Sensor_Correct_Position := NOT "AlwaysFALSE" AND ("Simu_Eleveytor" = 80);
   "DB_Data".F10.Position := NOT "AlwaysFALSE" AND ("Simu_Eleveytor" >= 90) AND ("Simu_Eleveytor" < 100);
   "DB_Data".F10.Sensor_Correct_Position := NOT "AlwaysFALSE" AND ("Simu_Eleveytor" = 90);
   "DB_Data".F11.Position := NOT "AlwaysFALSE" AND ("Simu_Eleveytor" >= 100) AND ("Simu_Eleveytor" < 110);
   "DB_Data".F11.Sensor_Correct_Position := NOT "AlwaysFALSE" AND ("Simu_Eleveytor" = 100);
   "DB_Data".F12.Position := NOT "AlwaysFALSE" AND ("Simu_Eleveytor" >= 110) AND ("Simu_Eleveytor" < 120);
   "DB_Data".F12.Sensor_Correct_Position := NOT "AlwaysFALSE" AND ("Simu_Eleveytor" = 110);
   "DB_Data".F13.Position := NOT "AlwaysFALSE" AND ("Simu_Eleveytor" >= 120) AND ("Simu_Eleveytor" < 130);
   "DB_Data".F13.Sensor_Correct_Position := NOT "AlwaysFALSE" AND ("Simu_Eleveytor" = 120);
   "DB_Data".F14.Position := NOT "AlwaysFALSE" AND ("Simu_Eleveytor" >= 130) AND ("Simu_Eleveytor" < 140);
   "DB_Data".F14.Sensor_Correct_Position := NOT "AlwaysFALSE" AND ("Simu_Eleveytor" = 130);
   "DB_Data".F15.Position := NOT "AlwaysFALSE" AND ("Simu_Eleveytor" >= 140) AND ("Simu_Eleveytor" < 150);
   "DB_Data".F15.Sensor_Correct_Position := NOT "AlwaysFALSE" AND ("Simu_Eleveytor" = 140);
   "DB_Data".F16.Position := NOT "AlwaysFALSE" AND ("Simu_Eleveytor" >= 150) AND ("Simu_Eleveytor" < 160);
   "DB_Data".F16.Sensor_Correct_Position := NOT "AlwaysFALSE" AND ("Simu_Eleveytor" = 150);
   "DB_Data".F17.Position := NOT "AlwaysFALSE" AND ("Simu_Eleveytor" >= 160) AND ("Simu_Eleveytor" < 170);
   "DB_Data".F17.Sensor_Correct_Position := NOT "AlwaysFALSE" AND ("Simu_Eleveytor" = 160);
   "DB_Data".F18.Position := NOT "AlwaysFALSE" AND ("Simu_Eleveytor" >= 170) AND ("Simu_Eleveytor" < 180);
   "DB_Data".F18.Sensor_Correct_Position := NOT "AlwaysFALSE" AND ("Simu_Eleveytor" = 170);
   "DB_Data".F19.Position := NOT "AlwaysFALSE" AND ("Simu_Eleveytor" >= 180) AND ("Simu_Eleveytor" < 190);
   "DB_Data".F19.Sensor_Correct_Position := NOT "AlwaysFALSE" AND ("Simu_Eleveytor" = 180);
   "DB_Data".F20.Position := NOT "AlwaysFALSE" AND ("Simu_Eleveytor" >= 190);
   "DB_Data".F20.Sensor_Correct_Position := NOT "AlwaysFALSE" AND ("Simu_Eleveytor" = 190);
END_REGION

REGION Network 3: Cửa buồng thang F1
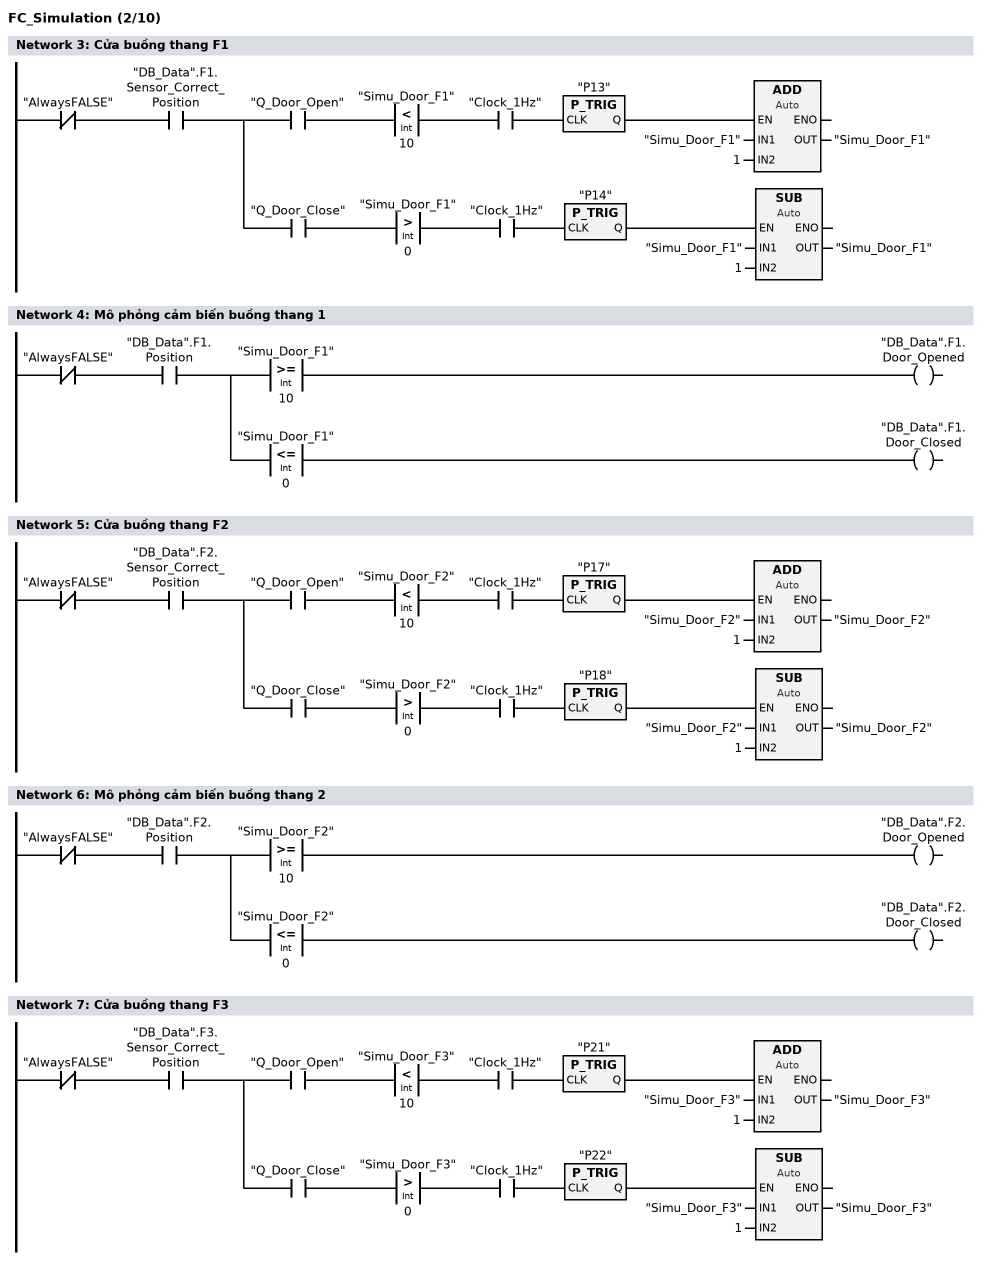
   RUNG wire#powerrail
      I_Contact( "AlwaysFALSE" )
      Contact( "DB_Data".F1.Sensor_Correct_Position )
      wire#w1
      Contact( "Q_Door_Open" )
      { S7_Templates := "SrcType := Int" } LT_Contact(in1 := "Simu_Door_F1", in2 := 10)
      Contact( "Clock_1Hz" )
      P_Trig( "P13" )
      Add(in1 := "Simu_Door_F1", in2 := 1, out => "Simu_Door_F1")
   END_RUNG
   RUNG wire#w1
      Contact( "Q_Door_Close" )
      { S7_Templates := "SrcType := Int" } GT_Contact(in1 := "Simu_Door_F1", in2 := 0)
      Contact( "Clock_1Hz" )
      P_Trig( "P14" )
      Sub(in1 := "Simu_Door_F1", in2 := 1, out => "Simu_Door_F1")
   END_RUNG
   // the same network as SCL:
   #_w1 := NOT "AlwaysFALSE" AND "DB_Data".F1.Sensor_Correct_Position;
   #_w2 := #_w1 AND "Q_Door_Open" AND ("Simu_Door_F1" < 10) AND "Clock_1Hz";
   #_w3 := #_w2 AND NOT "P13";   // rising edge
   "P13" := #_w2;
   IF #_w3 THEN "Simu_Door_F1" := "Simu_Door_F1" + 1; END_IF;
   #_w4 := #_w1 AND "Q_Door_Close" AND ("Simu_Door_F1" > 0) AND "Clock_1Hz";
   #_w5 := #_w4 AND NOT "P14";   // rising edge
   "P14" := #_w4;
   IF #_w5 THEN "Simu_Door_F1" := "Simu_Door_F1" - 1; END_IF;
END_REGION

REGION Network 4: Mô phỏng cảm biến buồng thang 1
   RUNG wire#powerrail
      I_Contact( "AlwaysFALSE" )
      Contact( "DB_Data".F1.Position )
      wire#w1
      { S7_Templates := "SrcType := Int" } GE_Contact(in1 := "Simu_Door_F1", in2 := 10)
      Coil( "DB_Data".F1.Door_Opened )
   END_RUNG
   RUNG wire#w1
      { S7_Templates := "SrcType := Int" } LE_Contact(in1 := "Simu_Door_F1", in2 := 0)
      Coil( "DB_Data".F1.Door_Closed )
   END_RUNG
   // the same network as SCL:
   #_w1 := NOT "AlwaysFALSE" AND "DB_Data".F1.Position;
   "DB_Data".F1.Door_Opened := #_w1 AND ("Simu_Door_F1" >= 10);
   "DB_Data".F1.Door_Closed := #_w1 AND ("Simu_Door_F1" <= 0);
END_REGION

REGION Network 5: Cửa buồng thang F2
   RUNG wire#powerrail
      I_Contact( "AlwaysFALSE" )
      Contact( "DB_Data".F2.Sensor_Correct_Position )
      wire#w1
      Contact( "Q_Door_Open" )
      { S7_Templates := "SrcType := Int" } LT_Contact(in1 := "Simu_Door_F2", in2 := 10)
      Contact( "Clock_1Hz" )
      P_Trig( "P17" )
      Add(in1 := "Simu_Door_F2", in2 := 1, out => "Simu_Door_F2")
   END_RUNG
   RUNG wire#w1
      Contact( "Q_Door_Close" )
      { S7_Templates := "SrcType := Int" } GT_Contact(in1 := "Simu_Door_F2", in2 := 0)
      Contact( "Clock_1Hz" )
      P_Trig( "P18" )
      Sub(in1 := "Simu_Door_F2", in2 := 1, out => "Simu_Door_F2")
   END_RUNG
   // the same network as SCL:
   #_w1 := NOT "AlwaysFALSE" AND "DB_Data".F2.Sensor_Correct_Position;
   #_w2 := #_w1 AND "Q_Door_Open" AND ("Simu_Door_F2" < 10) AND "Clock_1Hz";
   #_w3 := #_w2 AND NOT "P17";   // rising edge
   "P17" := #_w2;
   IF #_w3 THEN "Simu_Door_F2" := "Simu_Door_F2" + 1; END_IF;
   #_w4 := #_w1 AND "Q_Door_Close" AND ("Simu_Door_F2" > 0) AND "Clock_1Hz";
   #_w5 := #_w4 AND NOT "P18";   // rising edge
   "P18" := #_w4;
   IF #_w5 THEN "Simu_Door_F2" := "Simu_Door_F2" - 1; END_IF;
END_REGION

REGION Network 6: Mô phỏng cảm biến buồng thang 2
   RUNG wire#powerrail
      I_Contact( "AlwaysFALSE" )
      Contact( "DB_Data".F2.Position )
      wire#w1
      { S7_Templates := "SrcType := Int" } GE_Contact(in1 := "Simu_Door_F2", in2 := 10)
      Coil( "DB_Data".F2.Door_Opened )
   END_RUNG
   RUNG wire#w1
      { S7_Templates := "SrcType := Int" } LE_Contact(in1 := "Simu_Door_F2", in2 := 0)
      Coil( "DB_Data".F2.Door_Closed )
   END_RUNG
   // the same network as SCL:
   #_w1 := NOT "AlwaysFALSE" AND "DB_Data".F2.Position;
   "DB_Data".F2.Door_Opened := #_w1 AND ("Simu_Door_F2" >= 10);
   "DB_Data".F2.Door_Closed := #_w1 AND ("Simu_Door_F2" <= 0);
END_REGION

REGION Network 7: Cửa buồng thang F3
   RUNG wire#powerrail
      I_Contact( "AlwaysFALSE" )
      Contact( "DB_Data".F3.Sensor_Correct_Position )
      wire#w1
      Contact( "Q_Door_Open" )
      { S7_Templates := "SrcType := Int" } LT_Contact(in1 := "Simu_Door_F3", in2 := 10)
      Contact( "Clock_1Hz" )
      P_Trig( "P21" )
      Add(in1 := "Simu_Door_F3", in2 := 1, out => "Simu_Door_F3")
   END_RUNG
   RUNG wire#w1
      Contact( "Q_Door_Close" )
      { S7_Templates := "SrcType := Int" } GT_Contact(in1 := "Simu_Door_F3", in2 := 0)
      Contact( "Clock_1Hz" )
      P_Trig( "P22" )
      Sub(in1 := "Simu_Door_F3", in2 := 1, out => "Simu_Door_F3")
   END_RUNG
   // the same network as SCL:
   #_w1 := NOT "AlwaysFALSE" AND "DB_Data".F3.Sensor_Correct_Position;
   #_w2 := #_w1 AND "Q_Door_Open" AND ("Simu_Door_F3" < 10) AND "Clock_1Hz";
   #_w3 := #_w2 AND NOT "P21";   // rising edge
   "P21" := #_w2;
   IF #_w3 THEN "Simu_Door_F3" := "Simu_Door_F3" + 1; END_IF;
   #_w4 := #_w1 AND "Q_Door_Close" AND ("Simu_Door_F3" > 0) AND "Clock_1Hz";
   #_w5 := #_w4 AND NOT "P22";   // rising edge
   "P22" := #_w4;
   IF #_w5 THEN "Simu_Door_F3" := "Simu_Door_F3" - 1; END_IF;
END_REGION

REGION Network 8: Mô phỏng cảm biến buồng thang 3
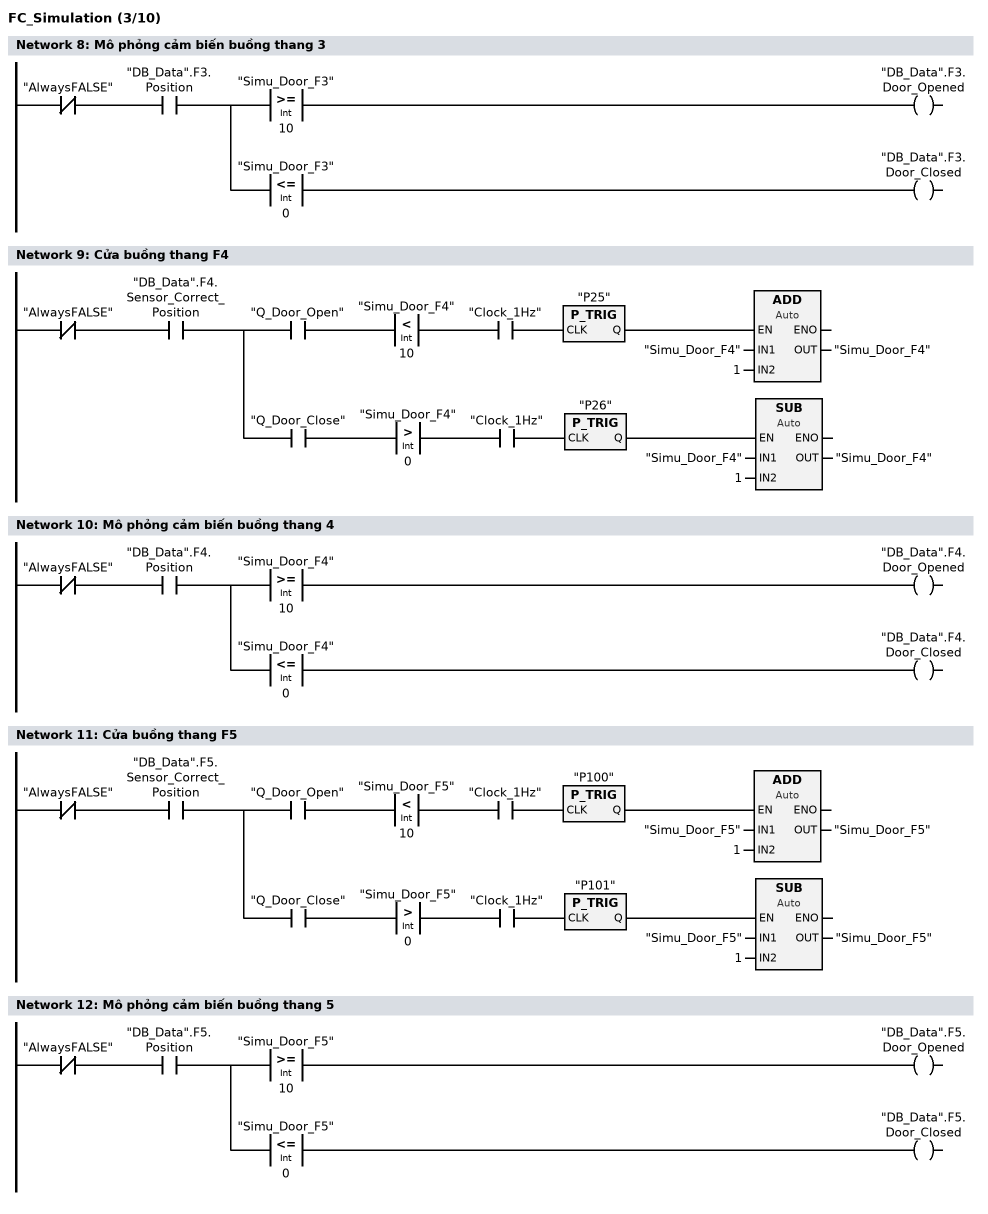
   RUNG wire#powerrail
      I_Contact( "AlwaysFALSE" )
      Contact( "DB_Data".F3.Position )
      wire#w1
      { S7_Templates := "SrcType := Int" } GE_Contact(in1 := "Simu_Door_F3", in2 := 10)
      Coil( "DB_Data".F3.Door_Opened )
   END_RUNG
   RUNG wire#w1
      { S7_Templates := "SrcType := Int" } LE_Contact(in1 := "Simu_Door_F3", in2 := 0)
      Coil( "DB_Data".F3.Door_Closed )
   END_RUNG
   // the same network as SCL:
   #_w1 := NOT "AlwaysFALSE" AND "DB_Data".F3.Position;
   "DB_Data".F3.Door_Opened := #_w1 AND ("Simu_Door_F3" >= 10);
   "DB_Data".F3.Door_Closed := #_w1 AND ("Simu_Door_F3" <= 0);
END_REGION

REGION Network 9: Cửa buồng thang F4
   RUNG wire#powerrail
      I_Contact( "AlwaysFALSE" )
      Contact( "DB_Data".F4.Sensor_Correct_Position )
      wire#w1
      Contact( "Q_Door_Open" )
      { S7_Templates := "SrcType := Int" } LT_Contact(in1 := "Simu_Door_F4", in2 := 10)
      Contact( "Clock_1Hz" )
      P_Trig( "P25" )
      Add(in1 := "Simu_Door_F4", in2 := 1, out => "Simu_Door_F4")
   END_RUNG
   RUNG wire#w1
      Contact( "Q_Door_Close" )
      { S7_Templates := "SrcType := Int" } GT_Contact(in1 := "Simu_Door_F4", in2 := 0)
      Contact( "Clock_1Hz" )
      P_Trig( "P26" )
      Sub(in1 := "Simu_Door_F4", in2 := 1, out => "Simu_Door_F4")
   END_RUNG
   // the same network as SCL:
   #_w1 := NOT "AlwaysFALSE" AND "DB_Data".F4.Sensor_Correct_Position;
   #_w2 := #_w1 AND "Q_Door_Open" AND ("Simu_Door_F4" < 10) AND "Clock_1Hz";
   #_w3 := #_w2 AND NOT "P25";   // rising edge
   "P25" := #_w2;
   IF #_w3 THEN "Simu_Door_F4" := "Simu_Door_F4" + 1; END_IF;
   #_w4 := #_w1 AND "Q_Door_Close" AND ("Simu_Door_F4" > 0) AND "Clock_1Hz";
   #_w5 := #_w4 AND NOT "P26";   // rising edge
   "P26" := #_w4;
   IF #_w5 THEN "Simu_Door_F4" := "Simu_Door_F4" - 1; END_IF;
END_REGION

REGION Network 10: Mô phỏng cảm biến buồng thang 4
   RUNG wire#powerrail
      I_Contact( "AlwaysFALSE" )
      Contact( "DB_Data".F4.Position )
      wire#w1
      { S7_Templates := "SrcType := Int" } GE_Contact(in1 := "Simu_Door_F4", in2 := 10)
      Coil( "DB_Data".F4.Door_Opened )
   END_RUNG
   RUNG wire#w1
      { S7_Templates := "SrcType := Int" } LE_Contact(in1 := "Simu_Door_F4", in2 := 0)
      Coil( "DB_Data".F4.Door_Closed )
   END_RUNG
   // the same network as SCL:
   #_w1 := NOT "AlwaysFALSE" AND "DB_Data".F4.Position;
   "DB_Data".F4.Door_Opened := #_w1 AND ("Simu_Door_F4" >= 10);
   "DB_Data".F4.Door_Closed := #_w1 AND ("Simu_Door_F4" <= 0);
END_REGION

REGION Network 11: Cửa buồng thang F5
   RUNG wire#powerrail
      I_Contact( "AlwaysFALSE" )
      Contact( "DB_Data".F5.Sensor_Correct_Position )
      wire#w1
      Contact( "Q_Door_Open" )
      { S7_Templates := "SrcType := Int" } LT_Contact(in1 := "Simu_Door_F5", in2 := 10)
      Contact( "Clock_1Hz" )
      P_Trig( "P100" )
      Add(in1 := "Simu_Door_F5", in2 := 1, out => "Simu_Door_F5")
   END_RUNG
   RUNG wire#w1
      Contact( "Q_Door_Close" )
      { S7_Templates := "SrcType := Int" } GT_Contact(in1 := "Simu_Door_F5", in2 := 0)
      Contact( "Clock_1Hz" )
      P_Trig( "P101" )
      Sub(in1 := "Simu_Door_F5", in2 := 1, out => "Simu_Door_F5")
   END_RUNG
   // the same network as SCL:
   #_w1 := NOT "AlwaysFALSE" AND "DB_Data".F5.Sensor_Correct_Position;
   #_w2 := #_w1 AND "Q_Door_Open" AND ("Simu_Door_F5" < 10) AND "Clock_1Hz";
   #_w3 := #_w2 AND NOT "P100";   // rising edge
   "P100" := #_w2;
   IF #_w3 THEN "Simu_Door_F5" := "Simu_Door_F5" + 1; END_IF;
   #_w4 := #_w1 AND "Q_Door_Close" AND ("Simu_Door_F5" > 0) AND "Clock_1Hz";
   #_w5 := #_w4 AND NOT "P101";   // rising edge
   "P101" := #_w4;
   IF #_w5 THEN "Simu_Door_F5" := "Simu_Door_F5" - 1; END_IF;
END_REGION

REGION Network 12: Mô phỏng cảm biến buồng thang 5
   RUNG wire#powerrail
      I_Contact( "AlwaysFALSE" )
      Contact( "DB_Data".F5.Position )
      wire#w1
      { S7_Templates := "SrcType := Int" } GE_Contact(in1 := "Simu_Door_F5", in2 := 10)
      Coil( "DB_Data".F5.Door_Opened )
   END_RUNG
   RUNG wire#w1
      { S7_Templates := "SrcType := Int" } LE_Contact(in1 := "Simu_Door_F5", in2 := 0)
      Coil( "DB_Data".F5.Door_Closed )
   END_RUNG
   // the same network as SCL:
   #_w1 := NOT "AlwaysFALSE" AND "DB_Data".F5.Position;
   "DB_Data".F5.Door_Opened := #_w1 AND ("Simu_Door_F5" >= 10);
   "DB_Data".F5.Door_Closed := #_w1 AND ("Simu_Door_F5" <= 0);
END_REGION

REGION Network 13: 6
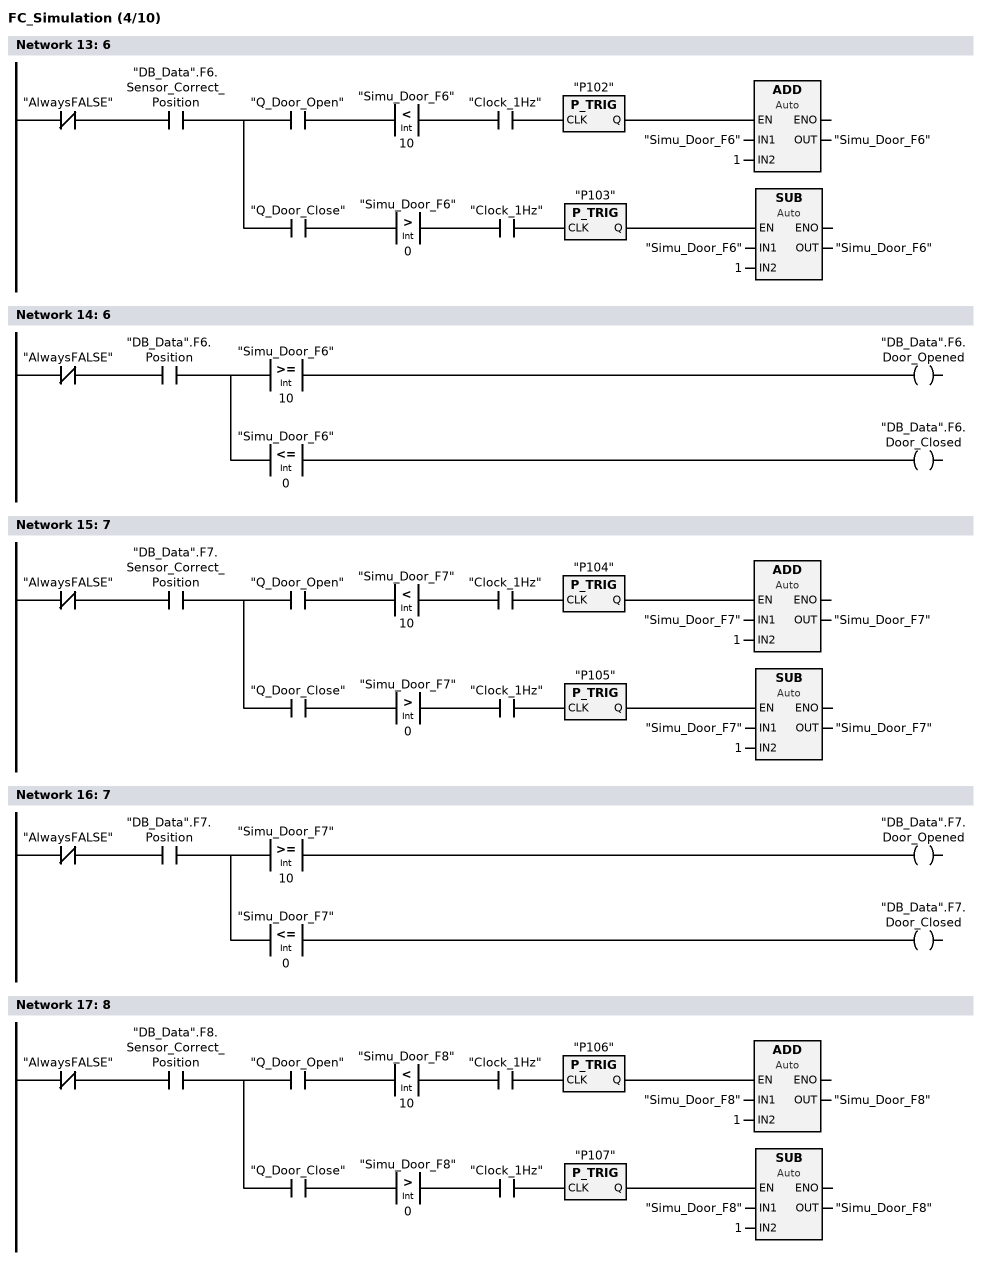
   RUNG wire#powerrail
      I_Contact( "AlwaysFALSE" )
      Contact( "DB_Data".F6.Sensor_Correct_Position )
      wire#w1
      Contact( "Q_Door_Open" )
      { S7_Templates := "SrcType := Int" } LT_Contact(in1 := "Simu_Door_F6", in2 := 10)
      Contact( "Clock_1Hz" )
      P_Trig( "P102" )
      Add(in1 := "Simu_Door_F6", in2 := 1, out => "Simu_Door_F6")
   END_RUNG
   RUNG wire#w1
      Contact( "Q_Door_Close" )
      { S7_Templates := "SrcType := Int" } GT_Contact(in1 := "Simu_Door_F6", in2 := 0)
      Contact( "Clock_1Hz" )
      P_Trig( "P103" )
      Sub(in1 := "Simu_Door_F6", in2 := 1, out => "Simu_Door_F6")
   END_RUNG
   // the same network as SCL:
   #_w1 := NOT "AlwaysFALSE" AND "DB_Data".F6.Sensor_Correct_Position;
   #_w2 := #_w1 AND "Q_Door_Open" AND ("Simu_Door_F6" < 10) AND "Clock_1Hz";
   #_w3 := #_w2 AND NOT "P102";   // rising edge
   "P102" := #_w2;
   IF #_w3 THEN "Simu_Door_F6" := "Simu_Door_F6" + 1; END_IF;
   #_w4 := #_w1 AND "Q_Door_Close" AND ("Simu_Door_F6" > 0) AND "Clock_1Hz";
   #_w5 := #_w4 AND NOT "P103";   // rising edge
   "P103" := #_w4;
   IF #_w5 THEN "Simu_Door_F6" := "Simu_Door_F6" - 1; END_IF;
END_REGION

REGION Network 14: 6
   RUNG wire#powerrail
      I_Contact( "AlwaysFALSE" )
      Contact( "DB_Data".F6.Position )
      wire#w1
      { S7_Templates := "SrcType := Int" } GE_Contact(in1 := "Simu_Door_F6", in2 := 10)
      Coil( "DB_Data".F6.Door_Opened )
   END_RUNG
   RUNG wire#w1
      { S7_Templates := "SrcType := Int" } LE_Contact(in1 := "Simu_Door_F6", in2 := 0)
      Coil( "DB_Data".F6.Door_Closed )
   END_RUNG
   // the same network as SCL:
   #_w1 := NOT "AlwaysFALSE" AND "DB_Data".F6.Position;
   "DB_Data".F6.Door_Opened := #_w1 AND ("Simu_Door_F6" >= 10);
   "DB_Data".F6.Door_Closed := #_w1 AND ("Simu_Door_F6" <= 0);
END_REGION

REGION Network 15: 7
   RUNG wire#powerrail
      I_Contact( "AlwaysFALSE" )
      Contact( "DB_Data".F7.Sensor_Correct_Position )
      wire#w1
      Contact( "Q_Door_Open" )
      { S7_Templates := "SrcType := Int" } LT_Contact(in1 := "Simu_Door_F7", in2 := 10)
      Contact( "Clock_1Hz" )
      P_Trig( "P104" )
      Add(in1 := "Simu_Door_F7", in2 := 1, out => "Simu_Door_F7")
   END_RUNG
   RUNG wire#w1
      Contact( "Q_Door_Close" )
      { S7_Templates := "SrcType := Int" } GT_Contact(in1 := "Simu_Door_F7", in2 := 0)
      Contact( "Clock_1Hz" )
      P_Trig( "P105" )
      Sub(in1 := "Simu_Door_F7", in2 := 1, out => "Simu_Door_F7")
   END_RUNG
   // the same network as SCL:
   #_w1 := NOT "AlwaysFALSE" AND "DB_Data".F7.Sensor_Correct_Position;
   #_w2 := #_w1 AND "Q_Door_Open" AND ("Simu_Door_F7" < 10) AND "Clock_1Hz";
   #_w3 := #_w2 AND NOT "P104";   // rising edge
   "P104" := #_w2;
   IF #_w3 THEN "Simu_Door_F7" := "Simu_Door_F7" + 1; END_IF;
   #_w4 := #_w1 AND "Q_Door_Close" AND ("Simu_Door_F7" > 0) AND "Clock_1Hz";
   #_w5 := #_w4 AND NOT "P105";   // rising edge
   "P105" := #_w4;
   IF #_w5 THEN "Simu_Door_F7" := "Simu_Door_F7" - 1; END_IF;
END_REGION

REGION Network 16: 7
   RUNG wire#powerrail
      I_Contact( "AlwaysFALSE" )
      Contact( "DB_Data".F7.Position )
      wire#w1
      { S7_Templates := "SrcType := Int" } GE_Contact(in1 := "Simu_Door_F7", in2 := 10)
      Coil( "DB_Data".F7.Door_Opened )
   END_RUNG
   RUNG wire#w1
      { S7_Templates := "SrcType := Int" } LE_Contact(in1 := "Simu_Door_F7", in2 := 0)
      Coil( "DB_Data".F7.Door_Closed )
   END_RUNG
   // the same network as SCL:
   #_w1 := NOT "AlwaysFALSE" AND "DB_Data".F7.Position;
   "DB_Data".F7.Door_Opened := #_w1 AND ("Simu_Door_F7" >= 10);
   "DB_Data".F7.Door_Closed := #_w1 AND ("Simu_Door_F7" <= 0);
END_REGION

REGION Network 17: 8
   RUNG wire#powerrail
      I_Contact( "AlwaysFALSE" )
      Contact( "DB_Data".F8.Sensor_Correct_Position )
      wire#w1
      Contact( "Q_Door_Open" )
      { S7_Templates := "SrcType := Int" } LT_Contact(in1 := "Simu_Door_F8", in2 := 10)
      Contact( "Clock_1Hz" )
      P_Trig( "P106" )
      Add(in1 := "Simu_Door_F8", in2 := 1, out => "Simu_Door_F8")
   END_RUNG
   RUNG wire#w1
      Contact( "Q_Door_Close" )
      { S7_Templates := "SrcType := Int" } GT_Contact(in1 := "Simu_Door_F8", in2 := 0)
      Contact( "Clock_1Hz" )
      P_Trig( "P107" )
      Sub(in1 := "Simu_Door_F8", in2 := 1, out => "Simu_Door_F8")
   END_RUNG
   // the same network as SCL:
   #_w1 := NOT "AlwaysFALSE" AND "DB_Data".F8.Sensor_Correct_Position;
   #_w2 := #_w1 AND "Q_Door_Open" AND ("Simu_Door_F8" < 10) AND "Clock_1Hz";
   #_w3 := #_w2 AND NOT "P106";   // rising edge
   "P106" := #_w2;
   IF #_w3 THEN "Simu_Door_F8" := "Simu_Door_F8" + 1; END_IF;
   #_w4 := #_w1 AND "Q_Door_Close" AND ("Simu_Door_F8" > 0) AND "Clock_1Hz";
   #_w5 := #_w4 AND NOT "P107";   // rising edge
   "P107" := #_w4;
   IF #_w5 THEN "Simu_Door_F8" := "Simu_Door_F8" - 1; END_IF;
END_REGION

REGION Network 18: 8
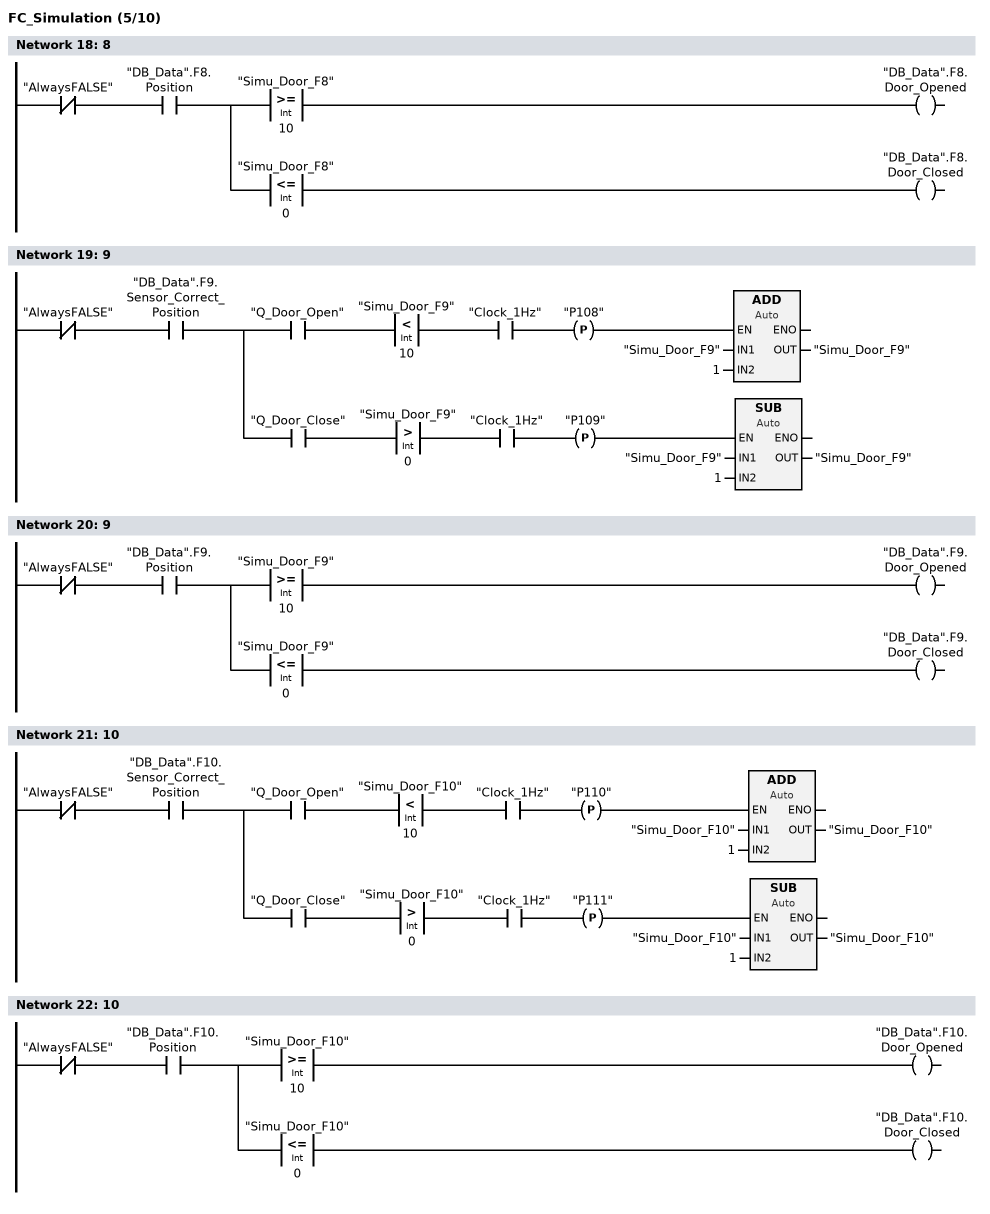
   RUNG wire#powerrail
      I_Contact( "AlwaysFALSE" )
      Contact( "DB_Data".F8.Position )
      wire#w1
      { S7_Templates := "SrcType := Int" } GE_Contact(in1 := "Simu_Door_F8", in2 := 10)
      Coil( "DB_Data".F8.Door_Opened )
   END_RUNG
   RUNG wire#w1
      { S7_Templates := "SrcType := Int" } LE_Contact(in1 := "Simu_Door_F8", in2 := 0)
      Coil( "DB_Data".F8.Door_Closed )
   END_RUNG
   // the same network as SCL:
   #_w1 := NOT "AlwaysFALSE" AND "DB_Data".F8.Position;
   "DB_Data".F8.Door_Opened := #_w1 AND ("Simu_Door_F8" >= 10);
   "DB_Data".F8.Door_Closed := #_w1 AND ("Simu_Door_F8" <= 0);
END_REGION

